C05467=1049.152,167.646,409.024,171.137,36.035,156.777
C05468=1049.158,167.895,409.001,171.139,36.037,156.778
C05469=1049.163,168.144,408.978,171.141,36.039,156.778
C05470=1049.169,168.392,408.955,171.143,36.041,156.778
C05471=1049.176,168.641,408.932,171.145,36.043,156.779
C05472=1049.181,168.890,408.909,171.148,36.046,156.779
C05473=1049.187,169.139,408.886,171.150,36.047,156.780
C05474=1049.194,169.388,408.862,171.152,36.050,156.780
C05475=1049.199,169.637,408.839,171.154,36.052,156.780
C05476=1049.205,169.886,408.817,171.157,36.054,156.781
C05477=1049.212,170.134,408.794,171.159,36.056,156.781
C05478=1049.217,170.383,408.771,171.161,36.058,156.782
C05479=1049.223,170.632,408.748,171.163,36.060,156.782
C05480=1049.229,170.881,408.725,171.165,36.062,156.783
C05481=1049.235,171.131,408.702,171.168,36.065,156.783
C05482=1049.241,171.379,408.678,171.170,36.067,156.783
C05483=1049.248,171.627,408.656,171.172,36.069,156.784
C05484=1049.253,171.876,408.633,171.174,36.071,156.784
C05485=1049.259,172.125,408.610,171.176,36.073,156.785
C05486=1049.265,172.374,408.587,171.179,36.075,156.785
C05487=1049.271,172.624,408.564,171.181,36.077,156.785
C05488=1049.277,172.872,408.540,171.183,36.080,156.786
C05489=1049.283,173.121,408.517,171.185,36.081,156.786
C05490=1049.289,173.369,408.495,171.188,36.084,156.787
C05491=1049.296,173.654,408.468,171.190,36.086,156.787
C05492=1049.303,173.939,408.442,171.193,36.089,156.788
C05493=1049.310,174.224,408.415,171.195,36.091,156.788
C05494=1049.317,174.508,408.388,171.198,36.094,156.789
C05495=1049.324,174.758,408.366,171.200,36.096,156.789
C05496=1049.329,175.007,408.343,171.202,36.097,156.789
C05497=1049.335,175.255,408.319,171.204,36.100,156.790
C05498=1049.341,175.504,408.296,171.206,36.102,156.790
C05499=1049.347,175.753,408.273,171.209,36.104,156.791
C05500=1049.353,176.002,408.249,171.211,36.106,156.791
C05501=1049.359,176.250,408.226,171.213,36.108,156.791
C05502=1049.365,176.499,408.203,171.216,36.110,156.792
C05503=1049.372,176.748,408.180,171.219,36.113,156.792
C05504=1049.378,176.997,408.157,171.221,36.115,156.793
C05505=1049.384,177.246,408.134,171.223,36.117,156.793
C05506=1049.390,177.495,408.110,171.225,36.119,156.794
C05507=1049.396,177.744,408.087,171.227,36.121,156.794
C05508=1049.402,177.992,408.063,171.230,36.123,156.794
C05509=1049.408,178.242,408.040,171.232,36.125,156.795
C05510=1049.414,178.490,408.017,171.234,36.128,156.795
C05511=1049.420,178.739,407.993,171.236,36.129,156.796
C05512=1049.427,178.988,407.970,171.239,36.132,156.796
C05513=1049.433,179.237,407.946,171.241,36.134,156.796
C05514=1049.439,179.485,407.924,171.243,36.136,156.797
C05515=1049.446,179.734,407.900,171.245,36.138,156.797
C05516=1049.451,179.983,407.877,171.247,36.140,156.798
C05517=1049.457,180.231,407.853,171.251,36.142,156.798
C05518=1049.464,180.481,407.830,171.253,36.145,156.799
C05519=1049.470,180.729,407.806,171.255,36.147,156.799
C05520=1049.476,180.979,407.783,171.257,36.149,156.799
C05521=1049.482,181.227,407.759,171.260,36.151,156.800
C05522=1049.488,181.476,407.736,171.262,36.153,156.800
C05523=1049.495,181.725,407.712,171.264,36.155,156.801
C05524=1049.501,181.973,407.689,171.266,36.158,156.801
C05525=1049.507,182.223,407.665,171.268,36.159,156.801
C05526=1049.513,182.471,407.642,171.272,36.162,156.802
C05527=1049.519,182.721,407.618,171.274,36.164,156.802
C05528=1049.526,182.969,407.595,171.276,36.166,156.803
C05529=1049.532,183.217,407.572,171.278,36.168,156.803
C05530=1049.538,183.467,407.548,171.281,36.170,156.804
C05531=1049.545,183.715,407.525,171.283,36.172,156.804
C05532=1049.551,183.964,407.501,171.285,36.175,156.804
C05533=1049.556,184.213,407.477,171.287,36.177,156.805
C05534=1049.563,184.462,407.453,171.290,36.179,156.805
C05535=1049.568,184.711,407.429,171.293,36.181,156.806
C05536=1049.574,184.959,407.405,171.295,36.184,156.806
C05537=1049.580,185.209,407.381,171.297,36.186,156.807
C05538=1049.586,185.457,407.358,171.300,36.188,156.807
C05539=1049.592,185.705,407.334,171.302,36.191,156.808
C05540=1049.598,185.955,407.309,171.304,36.193,156.808
C05541=1049.604,186.203,407.286,171.306,36.196,156.809
C05542=1049.609,186.451,407.261,171.309,36.197,156.809
C05543=1049.615,186.701,407.238,171.311,36.200,156.809
C05544=1049.621,186.950,407.214,171.313,36.202,156.810
C05545=1049.627,187.199,407.190,171.315,36.205,156.810
C05546=1049.633,187.447,407.166,171.319,36.207,156.811
C05547=1049.639,187.696,407.142,171.321,36.209,156.811
C05548=1049.645,187.945,407.117,171.323,36.211,156.812
C05549=1049.651,188.193,407.094,171.325,36.214,156.812
C05550=1049.656,188.442,407.069,171.328,36.216,156.813
C05551=1049.663,188.691,407.045,171.330,36.219,156.813
C05552=1049.668,188.940,407.021,171.332,36.221,156.814
C05553=1049.674,189.188,406.997,171.334,36.223,156.814
C05554=1049.680,189.438,406.972,171.338,36.226,156.815
C05555=1049.687,189.722,406.945,171.340,36.229,156.815
C05556=1049.694,190.006,406.918,171.342,36.231,156.816
C05557=1049.701,190.290,406.890,171.345,36.233,156.816
C05558=1049.708,190.575,406.863,171.348,36.236,156.817
C05559=1049.713,190.823,406.839,171.351,36.239,156.817
C05560=1049.720,191.072,406.815,171.353,36.241,156.818
C05561=1049.725,191.321,406.790,171.356,36.243,156.818
C05562=1049.732,191.570,406.766,171.358,36.246,156.819
C05563=1049.737,191.818,406.741,171.360,36.248,156.819
C05564=1049.744,192.067,406.717,171.362,36.251,156.820
C05565=1049.749,192.316,406.693,171.366,36.253,156.820
C05566=1049.756,192.564,406.669,171.368,36.255,156.820
C05567=1049.762,192.814,406.645,171.370,36.257,156.821
C05568=1049.768,193.062,406.621,171.372,36.260,156.821
C05569=1049.774,193.311,406.596,171.375,36.262,156.822
C05570=1049.779,193.560,406.572,171.377,36.265,156.822
C05571=1049.786,193.808,406.547,171.380,36.267,156.823
C05572=1049.791,194.057,406.523,171.382,36.269,156.823
C05573=1049.798,194.306,406.499,171.385,36.272,156.824
C05574=1049.804,194.555,406.474,171.387,36.274,156.824
C05575=1049.810,194.803,406.451,171.389,36.276,156.825
C05576=1049.816,195.052,406.425,171.392,36.279,156.825
C05577=1049.822,195.300,406.402,171.395,36.281,156.826
C05578=1049.828,195.550,406.377,171.397,36.283,156.826
C05579=1049.834,195.799,406.353,171.399,36.286,156.827
C05580=1049.840,196.047,406.328,171.402,36.288,156.827
C05581=1049.846,196.296,406.303,171.405,36.291,156.828
C05582=1049.853,196.545,406.279,171.407,36.293,156.828
C05583=1049.858,196.793,406.255,171.409,36.296,156.829
C05584=1049.865,197.042,406.230,171.412,36.297,156.829
C05585=1049.870,197.290,406.206,171.415,36.300,156.829
C05586=1049.877,197.539,406.182,171.417,36.302,156.830
C05587=1049.883,197.788,406.157,171.419,36.305,156.830
C05588=1049.889,198.037,406.132,171.422,36.307,156.831
C05589=1049.895,198.286,406.109,171.424,36.310,156.831
C05590=1049.901,198.534,406.083,171.427,36.312,156.832
C05591=1049.908,198.783,406.059,171.430,36.314,156.832
C05592=1049.913,199.031,406.034,171.432,36.317,156.833
C05593=1049.920,199.280,406.010,171.434,36.319,156.833
C05594=1049.926,199.530,405.986,171.437,36.322,156.834
C05595=1049.932,199.777,405.961,171.440,36.324,156.834
C05596=1049.938,200.026,405.937,171.442,36.327,156.835
C05597=1049.944,200.275,405.911,171.445,36.329,156.835
C05598=1049.951,200.524,405.887,171.447,36.331,156.836
C05599=1049.957,200.772,405.862,171.450,36.333,156.836
C05600=1049.962,201.021,405.838,171.452,36.336,156.837
C05601=1049.969,201.270,405.813,171.455,36.338,156.837
C05602=1049.975,201.519,405.788,171.458,36.341,156.838
C05603=1049.982,201.768,405.763,171.460,36.343,156.838
C05604=1049.987,202.016,405.739,171.462,36.346,156.839
C05605=1049.993,202.265,405.713,171.465,36.348,156.839
C05606=1050.000,202.514,405.689,171.468,36.351,156.840
C05607=1050.005,202.762,405.664,171.470,36.353,156.840
C05608=1050.011,203.011,405.639,171.472,36.356,156.841
C05609=1050.017,203.260,405.614,171.476,36.358,156.841
C05610=1050.024,203.509,405.589,171.478,36.361,156.842
C05611=1050.029,203.757,405.565,171.480,36.364,156.842
C05612=1050.035,204.006,405.539,171.483,36.366,156.843
C05613=1050.041,204.254,405.514,171.486,36.368,156.843
C05614=1050.048,204.503,405.489,171.488,36.371,156.844
C05615=1050.053,204.752,405.464,171.490,36.373,156.844
C05616=1050.059,205.000,405.439,171.494,36.376,156.845
C05617=1050.065,205.249,405.414,171.496,36.379,156.845
C05618=1050.072,205.498,405.390,171.498,36.381,156.846
C05619=1050.097,206.550,405.283,171.730,36.477,156.865
C05620=1050.104,206.804,405.256,171.731,36.481,156.866
C05621=1050.111,207.059,405.230,171.733,36.485,156.867
C05622=1050.118,207.314,405.204,171.736,36.488,156.867
C05623=1050.124,207.567,405.177,171.737,36.491,156.868
C05624=1050.131,207.816,405.150,171.740,36.495,156.869
C05625=1050.137,208.065,405.125,171.742,36.498,156.870
C05626=1050.143,208.313,405.098,171.744,36.501,156.870
C05627=1050.150,208.562,405.072,171.746,36.504,156.871
C05628=1050.156,208.811,405.046,171.747,36.508,156.872
C05629=1050.162,209.060,405.019,171.750,36.511,156.872
C05630=1050.169,209.308,404.993,171.751,36.515,156.873
C05631=1050.175,209.556,404.967,171.754,36.518,156.874
C05632=1050.182,209.805,404.940,171.756,36.521,156.874
C05633=1050.188,210.053,404.915,171.757,36.525,156.875
C05634=1050.194,210.301,404.889,171.760,36.528,156.876
C05635=1050.201,210.551,404.862,171.762,36.531,156.876
C05636=1050.207,210.799,404.836,171.764,36.534,156.877
C05637=1050.214,211.047,404.809,171.766,36.538,156.878
C05638=1050.220,211.296,404.783,171.767,36.541,156.878
C05639=1050.226,211.544,404.757,171.770,36.545,156.879
C05640=1050.233,211.793,404.730,171.772,36.548,156.880
C05641=1050.239,212.041,404.704,171.774,36.551,156.881
C05642=1050.246,212.290,404.678,171.776,36.554,156.881
C05643=1050.252,212.539,404.651,171.778,36.558,156.882
C05644=1050.258,212.787,404.625,171.780,36.561,156.883
C05645=1050.265,213.036,404.598,171.782,36.564,156.883
C05646=1050.271,213.284,404.571,171.784,36.568,156.884
C05647=1050.278,213.533,404.545,171.786,36.571,156.885
C05648=1050.284,213.781,404.518,171.789,36.575,156.885
C05649=1050.290,214.029,404.492,171.790,36.577,156.886
C05650=1050.297,214.278,404.465,171.792,36.581,156.887
C05651=1050.303,214.526,404.439,171.795,36.584,156.887
C05652=1050.310,214.775,404.412,171.796,36.588,156.888
C05653=1050.316,215.023,404.386,171.799,36.591,156.889
C05654=1050.322,215.272,404.359,171.801,36.594,156.890
C05655=1050.328,215.521,404.333,171.803,36.598,156.890
C05656=1050.335,215.770,404.306,171.805,36.601,156.891
C05657=1050.341,216.018,404.279,171.807,36.604,156.892
C05658=1050.348,216.266,404.253,171.809,36.607,156.892
C05659=1050.354,216.515,404.226,171.811,36.611,156.893
C05660=1050.360,216.763,404.200,171.814,36.614,156.894
C05661=1050.367,217.012,404.173,171.815,36.618,156.894
C05662=1050.373,217.260,404.146,171.817,36.621,156.895
C05663=1050.380,217.509,404.120,171.820,36.624,156.896
C05664=1050.386,217.757,404.093,171.821,36.627,156.896
C05665=1050.393,218.006,404.067,171.824,36.630,156.897
C05666=1050.399,218.255,404.039,171.826,36.634,156.898
C05667=1050.406,218.502,404.013,171.828,36.637,156.898
C05668=1050.413,218.751,403.986,171.830,36.640,156.899
C05669=1050.418,219.000,403.959,171.832,36.643,156.900
C05670=1050.425,219.248,403.933,171.835,36.647,156.901
C05671=1050.431,219.497,403.906,171.836,36.650,156.901
C05672=1050.439,219.745,403.879,171.839,36.653,156.902
C05673=1050.444,219.993,403.852,171.841,36.656,156.903
C05674=1050.451,220.242,403.825,171.842,36.659,156.903
C05675=1050.458,220.491,403.799,171.845,36.663,156.904
C05676=1050.464,220.751,403.771,171.847,36.667,156.905
C05677=1050.471,221.011,403.743,171.850,36.670,156.905
C05678=1050.478,221.271,403.714,171.852,36.673,156.906
C05679=1050.484,221.530,403.686,171.854,36.677,156.907
C05680=1050.491,221.779,403.659,171.856,36.680,156.907
C05681=1050.496,222.028,403.632,171.859,36.683,156.908
C05682=1050.503,222.276,403.604,171.861,36.686,156.909
C05683=1050.510,222.524,403.578,171.862,36.690,156.910
C05684=1050.516,222.773,403.550,171.865,36.693,156.910
C05685=1050.522,223.021,403.524,171.867,36.696,156.911
C05686=1050.528,223.270,403.497,171.869,36.699,156.912
C05687=1050.535,223.519,403.469,171.871,36.703,156.912
C05688=1050.541,223.767,403.442,171.874,36.706,156.913
C05689=1050.548,224.015,403.415,171.876,36.709,156.914
C05690=1050.554,224.263,403.389,171.877,36.712,156.914
C05691=1050.561,224.512,403.361,171.880,36.716,156.915
C05692=1050.567,224.761,403.334,171.882,36.719,156.916
C05693=1050.573,225.009,403.306,171.885,36.723,156.916
C05694=1050.580,225.258,403.279,171.887,36.726,156.917
C05695=1050.586,225.506,403.252,171.889,36.729,156.918
C05696=1050.592,225.755,403.225,171.891,36.732,156.918
C05697=1050.599,226.003,403.197,171.893,36.736,156.919
C05698=1050.606,226.252,403.171,171.896,36.739,156.920
C05699=1050.612,226.499,403.144,171.897,36.742,156.920
C05700=1050.618,226.749,403.117,171.900,36.745,156.921
C05701=1050.625,226.997,403.089,171.902,36.748,156.922
C05702=1050.631,227.245,403.061,171.905,36.752,156.923
C05703=1050.637,227.494,403.034,171.907,36.755,156.923
C05704=1050.644,227.742,403.007,171.908,36.758,156.924
C05705=1050.650,227.991,402.980,171.911,36.761,156.925
C05706=1050.657,228.239,402.952,171.913,36.764,156.925
C05707=1050.664,228.487,402.925,171.916,36.768,156.926
C05708=1050.670,228.736,402.898,171.918,36.771,156.927
C05709=1050.676,228.984,402.871,171.921,36.774,156.927
C05710=1050.683,229.232,402.843,171.922,36.777,156.928
C05711=1050.689,229.481,402.816,171.924,36.780,156.929
C05712=1050.695,229.729,402.788,171.927,36.784,156.929
C05713=1050.701,229.978,402.760,171.929,36.787,156.930
C05714=1050.708,230.226,402.733,171.932,36.790,156.931
C05715=1050.715,230.475,402.705,171.933,36.793,156.931
C05716=1050.721,230.723,402.678,171.936,36.797,156.932
C05717=1050.727,230.972,402.651,171.938,36.800,156.933
C05718=1050.734,231.220,402.623,171.941,36.804,156.934
C05719=1050.740,231.468,402.595,171.943,36.806,156.934
C05720=1050.747,231.716,402.568,171.945,36.809,156.935
C05721=1050.752,231.966,402.540,171.947,36.813,156.936
C05722=1050.759,232.214,402.512,171.949,36.816,156.936
C05723=1050.766,232.462,402.485,171.952,36.820,156.937
C05724=1050.772,232.710,402.457,171.954,36.823,156.938
C05725=1050.779,232.959,402.430,171.957,36.826,156.938
C05726=1050.785,233.207,402.402,171.959,36.829,156.939
C05727=1050.791,233.456,402.373,171.962,36.833,156.940
C05728=1050.797,233.704,402.346,171.963,36.836,156.940
C05729=1050.804,233.952,402.318,171.965,36.839,156.941
C05730=1050.811,234.200,402.291,171.968,36.842,156.942
C05731=1050.817,234.449,402.262,171.970,36.846,156.943
C05732=1050.823,234.702,402.235,171.973,36.849,156.943
C05733=1050.829,234.954,402.207,171.975,36.852,156.944
C05734=1050.836,235.206,402.178,171.978,36.855,156.945
C05735=1050.842,235.459,402.150,171.980,36.859,156.945
C05736=1050.849,235.707,402.122,171.982,36.862,156.946
C05737=1050.855,235.956,402.094,171.984,36.865,156.947
C05738=1050.862,236.204,402.066,171.986,36.868,156.947
C05739=1050.868,236.453,402.038,171.989,36.871,156.948
C05740=1050.874,236.701,402.011,171.991,36.875,156.949
C05741=1050.881,236.949,401.983,171.994,36.878,156.949
C05742=1050.887,237.198,401.955,171.996,36.881,156.950
C05743=1050.893,237.446,401.927,171.999,36.884,156.951
C05744=1050.900,237.695,401.899,172.001,36.888,156.951
C05745=1050.907,237.942,401.871,172.004,36.891,156.952
C05746=1050.913,238.191,401.842,172.006,36.894,156.953
C05747=1050.920,238.440,401.815,172.007,36.897,156.954
C05748=1050.926,238.687,401.787,172.010,36.900,156.954
C05749=1050.932,238.936,401.759,172.012,36.904,156.955
C05750=1050.938,239.185,401.731,172.015,36.907,156.956
C05751=1050.945,239.432,401.703,172.017,36.910,156.956
C05752=1050.951,239.681,401.675,172.020,36.913,156.957
C05753=1050.958,239.930,401.647,172.022,36.916,156.958
C05754=1050.965,240.178,401.619,172.025,36.920,156.958
C05755=1050.971,240.427,401.591,172.027,36.923,156.959
C05756=1050.977,240.675,401.562,172.029,36.926,156.960
C05757=1050.983,240.923,401.534,172.032,36.929,156.960
C05758=1050.990,241.172,401.506,172.034,36.932,156.961
C05759=1050.997,241.420,401.478,172.037,36.936,156.962
C05760=1051.003,241.668,401.450,172.039,36.939,156.962
C05761=1051.009,241.916,401.422,172.042,36.942,156.963
C05762=1051.015,242.164,401.393,172.044,36.945,156.964
C05763=1051.022,242.413,401.365,172.047,36.948,156.964
C05764=1051.028,242.661,401.337,172.049,36.952,156.965
C05765=1051.034,242.910,401.308,172.051,36.955,156.966
C05766=1051.041,243.158,401.280,172.053,36.958,156.967
C05767=1051.047,243.406,401.251,172.056,36.961,156.967
C05768=1051.054,243.655,401.224,172.058,36.965,156.968
C05769=1051.060,243.903,401.195,172.060,36.968,156.969
C05770=1051.066,244.151,401.166,172.063,36.971,156.969
C05771=1051.073,244.400,401.138,172.065,36.974,156.970
C05772=1051.079,244.648,401.109,172.068,36.978,156.971
C05773=1051.086,244.896,401.082,172.070,36.981,156.971
C05774=1051.092,245.145,401.053,172.073,36.984,156.972
C05775=1051.098,245.393,401.024,172.075,36.987,156.973
C05776=1051.105,245.641,400.996,172.078,36.990,156.973
C05777=1051.111,245.890,400.968,172.080,36.994,156.974
C05778=1051.117,246.138,400.938,172.083,36.996,156.975
C05779=1051.123,246.386,400.909,172.085,37.000,156.976
C05780=1051.130,246.635,400.882,172.088,37.004,156.976
C05781=1051.136,246.883,400.853,172.090,37.006,156.977
C05782=1051.142,247.131,400.824,172.093,37.010,156.978
C05783=1051.148,247.380,400.795,172.095,37.013,156.978
C05784=1051.155,247.628,400.766,172.097,37.017,156.979
C05785=1051.161,247.876,400.737,172.100,37.019,156.980
C05786=1051.168,248.124,400.709,172.102,37.023,156.981
C05787=1051.174,248.372,400.680,172.105,37.026,156.981
C05788=1051.179,248.620,400.652,172.107,37.029,156.982
C05789=1051.186,248.867,400.624,172.110,37.032,156.983
C05790=1051.192,249.114,400.594,172.112,37.036,156.983
C05791=1051.198,249.362,400.565,172.115,37.039,156.984
C05792=1051.204,249.609,400.537,172.117,37.042,156.985
C05793=1051.211,249.857,400.508,172.120,37.045,156.985
C05794=1051.217,250.104,400.480,172.122,37.049,156.986
C05795=1051.224,250.352,400.450,172.125,37.052,156.987
C05796=1051.230,250.600,400.421,172.127,37.055,156.988
C05797=1051.236,250.849,400.393,172.131,37.058,156.988
C05798=1051.243,251.096,400.364,172.133,37.062,156.989
C05799=1051.249,251.345,400.335,172.136,37.065,156.990
C05800=1051.255,251.593,400.306,172.138,37.068,156.990
C05801=1051.262,251.841,400.277,172.140,37.071,156.991
C05802=1051.268,252.089,400.248,172.143,37.075,156.992
C05803=1051.274,252.337,400.219,172.145,37.078,156.993
C05804=1051.281,252.587,400.191,172.148,37.081,156.993
C05805=1051.287,252.835,400.162,172.150,37.084,156.994
C05806=1051.293,253.083,400.133,172.153,37.088,156.995
C05807=1051.300,253.331,400.104,172.155,37.091,156.995
C05808=1051.306,253.579,400.075,172.158,37.094,156.996
C05809=1051.313,253.827,400.046,172.160,37.097,156.997
C05810=1051.319,254.075,400.017,172.164,37.101,156.998
C05811=1051.326,254.324,399.988,172.166,37.104,156.998
C05812=1051.332,254.572,399.959,172.169,37.107,156.999
C05813=1051.338,254.820,399.929,172.171,37.110,157.000
C05814=1051.344,255.068,399.900,172.174,37.114,157.000
C05815=1051.351,255.316,399.871,172.176,37.116,157.001
C05816=1051.358,255.565,399.842,172.179,37.119,157.002
C05817=1051.364,255.813,399.813,172.181,37.123,157.002
C05818=1051.370,256.061,399.784,172.184,37.126,157.003
C05819=1051.377,256.309,399.755,172.187,37.129,157.004
C05820=1051.384,256.558,399.725,172.190,37.132,157.004
C05821=1051.390,256.806,399.696,172.192,37.136,157.005
C05822=1051.397,257.054,399.667,172.195,37.139,157.006
C05823=1051.403,257.302,399.638,172.197,37.142,157.007
C05824=1051.410,257.551,399.609,172.200,37.145,157.007
C05825=1051.416,257.799,399.580,172.202,37.148,157.008
C05826=1051.422,258.047,399.551,172.205,37.152,157.009
C05827=1051.429,258.295,399.521,172.208,37.155,157.009
C05828=1051.436,258.543,399.492,172.210,37.158,157.010
C05829=1051.442,258.791,399.463,172.213,37.161,157.011
C05830=1051.448,259.040,399.433,172.215,37.165,157.012
C05831=1051.455,259.288,399.404,172.218,37.167,157.012
C05832=1051.462,259.536,399.374,172.221,37.171,157.013
C05833=1051.468,259.784,399.345,172.224,37.174,157.014
C05834=1051.475,260.033,399.316,172.226,37.177,157.014
C05835=1051.481,260.281,399.287,172.229,37.180,157.015
C05836=1051.488,260.529,399.257,172.231,37.183,157.016
C05837=1051.494,260.777,399.228,172.235,37.187,157.016
C05838=1051.501,261.026,399.199,172.237,37.190,157.017
C05839=1051.507,261.273,399.169,172.240,37.193,157.018
C05840=1051.514,261.522,399.139,172.242,37.196,157.019
C05841=1051.520,261.770,399.110,172.245,37.199,157.019
C05842=1051.527,262.018,399.080,172.248,37.203,157.020
C05843=1051.534,262.266,399.051,172.251,37.205,157.021
C05844=1051.540,262.513,399.022,172.253,37.208,157.021
C05845=1051.547,262.759,398.993,172.256,37.212,157.022
C05846=1051.553,263.005,398.964,172.259,37.215,157.023
C05847=1051.559,263.252,398.934,172.262,37.218,157.023
C05848=1051.566,263.498,398.905,172.264,37.221,157.024
C05849=1051.573,263.746,398.875,172.267,37.225,157.025
C05850=1051.579,263.992,398.846,172.269,37.228,157.026
C05851=1051.585,264.239,398.815,172.273,37.231,157.026
C05852=1051.591,264.487,398.786,172.275,37.235,157.027
C05853=1051.598,264.734,398.757,172.278,37.238,157.028
C05854=1051.604,264.983,398.726,172.280,37.241,157.028
C05855=1051.611,265.231,398.697,172.283,37.244,157.029
C05856=1051.618,265.479,398.667,172.286,37.247,157.030
C05857=1051.623,265.728,398.637,172.289,37.250,157.031
C05858=1051.630,265.975,398.607,172.291,37.254,157.031
C05859=1051.637,266.223,398.577,172.294,37.257,157.032
C05860=1051.642,266.472,398.548,172.297,37.260,157.033
C05861=1051.650,266.720,398.517,172.300,37.264,157.034
C05862=1051.656,266.967,398.488,172.302,37.267,157.034
C05863=1051.662,267.217,398.458,172.305,37.270,157.035
C05864=1051.669,267.464,398.428,172.308,37.273,157.036
C05865=1051.675,267.712,398.398,172.311,37.277,157.036
C05866=1051.682,267.960,398.367,172.313,37.280,157.037
C05867=1051.688,268.208,398.338,172.316,37.283,157.038
C05868=1051.694,268.457,398.308,172.319,37.286,157.039
C05869=1051.701,268.704,398.278,172.322,37.289,157.039
C05870=1051.707,268.953,398.247,172.324,37.293,157.040
C05871=1051.714,269.200,398.217,172.328,37.296,157.041
C05872=1051.720,269.449,398.187,172.330,37.299,157.041
C05873=1051.727,269.697,398.158,172.333,37.303,157.042
C05874=1051.733,269.945,398.127,172.335,37.306,157.043
C05875=1051.740,270.193,398.097,172.339,37.309,157.044
C05876=1051.746,270.442,398.067,172.341,37.313,157.044
C05877=1051.753,270.689,398.037,172.344,37.316,157.045
C05878=1051.759,270.938,398.006,172.347,37.319,157.046
C05879=1051.766,271.185,397.976,172.350,37.322,157.047
C05880=1051.772,271.434,397.946,172.353,37.325,157.047
C05881=1051.779,271.681,397.916,172.356,37.329,157.048
C05882=1051.785,271.930,397.885,172.359,37.332,157.049
C05883=1051.792,272.177,397.855,172.361,37.335,157.049
C05884=1051.798,272.426,397.825,172.365,37.339,157.050
C05885=1051.804,272.673,397.794,172.367,37.342,157.051
C05886=1051.811,272.922,397.764,172.370,37.345,157.052
C05887=1051.817,273.169,397.734,172.373,37.349,157.052
C05888=1051.823,273.418,397.703,172.376,37.352,157.053
C05889=1051.830,273.666,397.673,172.378,37.355,157.054
C05890=1051.836,273.914,397.643,172.382,37.359,157.055
C05891=1051.843,274.163,397.612,172.384,37.361,157.055
C05892=1051.849,274.410,397.582,172.387,37.365,157.056
C05893=1051.856,274.659,397.551,172.390,37.368,157.057
C05894=1051.861,274.906,397.521,172.393,37.371,157.058
C05895=1051.869,275.154,397.490,172.395,37.375,157.058
C05896=1051.875,275.403,397.460,172.399,37.378,157.059
C05897=1051.881,275.650,397.429,172.401,37.381,157.060
C05898=1051.887,275.899,397.398,172.404,37.385,157.061
C05899=1051.894,276.146,397.368,172.408,37.388,157.061
C05900=1051.900,276.396,397.337,172.410,37.392,157.062
C05901=1051.907,276.644,397.306,172.414,37.394,157.063
C05902=1051.914,276.894,397.275,172.416,37.398,157.064
C05903=1051.920,277.143,397.245,172.419,37.401,157.064
C05904=1051.927,277.391,397.214,172.422,37.404,157.065
C05905=1051.933,277.639,397.183,172.425,37.408,157.066
C05906=1051.940,277.887,397.153,172.427,37.411,157.067
C05907=1051.946,278.135,397.123,172.431,37.415,157.067
C05908=1051.953,278.383,397.091,172.433,37.418,157.068
C05909=1051.959,278.631,397.061,172.437,37.421,157.069
C05910=1051.965,278.879,397.029,172.440,37.425,157.070
C05911=1051.972,279.127,396.999,172.442,37.427,157.070
C05912=1051.978,279.375,396.969,172.446,37.431,157.071
C05913=1051.985,279.623,396.938,172.448,37.434,157.072
C05914=1051.991,279.871,396.907,172.452,37.438,157.073
C05915=1051.997,280.119,396.876,172.454,37.441,157.073
C05916=1052.004,280.367,396.845,172.458,37.444,157.074
C05917=1052.011,280.615,396.814,172.460,37.448,157.075
C05918=1052.017,280.864,396.783,172.463,37.451,157.076
C05919=1052.023,281.111,396.752,172.467,37.455,157.076
C05920=1052.030,281.359,396.721,172.469,37.458,157.077
C05921=1052.036,281.607,396.690,172.473,37.461,157.078
C05922=1052.042,281.854,396.659,172.475,37.464,157.079
C05923=1052.049,282.103,396.628,172.479,37.468,157.079
C05924=1052.056,282.351,396.596,172.481,37.471,157.080
C05925=1052.062,282.599,396.566,172.484,37.475,157.081
C05926=1052.068,282.847,396.535,172.487,37.478,157.082
C05927=1052.075,283.094,396.503,172.490,37.481,157.082
C05928=1052.081,283.343,396.472,172.493,37.485,157.083
C05929=1052.088,283.591,396.441,172.496,37.488,157.084
C05930=1052.094,283.838,396.410,172.500,37.492,157.085
C05931=1052.101,284.086,396.379,172.502,37.495,157.086
C05932=1052.107,284.335,396.348,172.506,37.498,157.086
C05933=1052.114,284.582,396.316,172.508,37.501,157.087
C05934=1052.121,284.830,396.285,172.512,37.505,157.088
C05935=1052.127,285.078,396.254,172.514,37.508,157.089
C05936=1052.133,285.326,396.223,172.518,37.512,157.089
C05937=1052.139,285.574,396.191,172.521,37.515,157.090
C05938=1052.146,285.822,396.160,172.524,37.519,157.091
C05939=1052.153,286.070,396.128,172.527,37.522,157.092
C05940=1052.159,286.318,396.097,172.530,37.525,157.092
C05941=1052.165,286.566,396.067,172.533,37.528,157.093
C05942=1052.172,286.814,396.035,172.536,37.532,157.094
C05943=1052.179,287.062,396.004,172.539,37.535,157.095
C05944=1052.185,287.310,395.972,172.543,37.539,157.096
C05945=1052.192,287.557,395.941,172.545,37.542,157.096
C05946=1052.199,287.805,395.909,172.549,37.545,157.097
C05947=1052.206,288.053,395.878,172.551,37.549,157.098
C05948=1052.212,288.301,395.846,172.555,37.552,157.099
C05949=1052.218,288.549,395.814,172.557,37.555,157.099
C05950=1052.224,288.797,395.783,172.561,37.559,157.100
C05951=1052.231,289.044,395.752,172.564,37.562,157.101
C05952=1052.237,289.293,395.720,172.567,37.566,157.102
C05953=1052.244,289.541,395.689,172.570,37.569,157.103
C05954=1052.251,289.788,395.657,172.573,37.573,157.103
C05955=1052.257,290.036,395.626,172.577,37.576,157.104
C05956=1052.267,290.423,395.576,172.582,37.581,157.105
C05957=1052.277,290.809,395.527,172.587,37.587,157.107
C05958=1052.287,291.195,395.477,172.592,37.592,157.108
C05959=1052.297,291.581,395.427,172.597,37.597,157.109
C05960=1052.308,291.951,395.380,172.601,37.603,157.110
C05961=1052.317,292.321,395.333,172.605,37.608,157.111
C05962=1052.327,292.691,395.285,172.610,37.613,157.113
C05963=1052.337,293.061,395.238,172.615,37.618,157.114
C05964=1052.343,293.309,395.206,172.619,37.621,157.115
C05965=1052.350,293.557,395.174,172.621,37.625,157.115
C05966=1052.357,293.805,395.142,172.625,37.628,157.116
C05967=1052.363,294.053,395.110,172.628,37.632,157.117
C05968=1052.369,294.301,395.079,172.631,37.635,157.118
C05969=1052.376,294.548,395.046,172.635,37.639,157.119
C05970=1052.382,294.796,395.014,172.637,37.642,157.119
C05971=1052.389,295.044,394.982,172.641,37.646,157.120
C05972=1052.395,295.292,394.950,172.644,37.649,157.121
C05973=1052.402,295.540,394.919,172.647,37.653,157.122
C05974=1052.408,295.787,394.886,172.651,37.656,157.123
C05975=1052.415,296.035,394.855,172.654,37.660,157.124
C05976=1052.422,296.283,394.822,172.657,37.663,157.124
C05977=1052.427,296.531,394.790,172.661,37.667,157.125
C05978=1052.435,296.778,394.758,172.663,37.670,157.126
C05979=1052.441,297.026,394.725,172.667,37.674,157.127
C05980=1052.447,297.274,394.693,172.670,37.678,157.128
C05981=1052.453,297.522,394.660,172.673,37.681,157.128
C05982=1052.460,297.770,394.629,172.677,37.685,157.129
C05983=1052.466,298.017,394.596,172.680,37.688,157.130
C05984=1052.472,298.265,394.563,172.683,37.692,157.131
C05985=1052.478,298.513,394.531,172.687,37.695,157.132
C05986=1052.485,298.761,394.498,172.689,37.699,157.133
C05987=1052.492,299.009,394.466,172.693,37.703,157.134
C05988=1052.499,299.256,394.433,172.697,37.706,157.134
C05989=1052.505,299.504,394.401,172.699,37.709,157.135
C05990=1052.511,299.752,394.368,172.703,37.713,157.136
C05991=1052.517,300.000,394.336,172.707,37.717,157.137
C05992=1052.524,300.247,394.304,172.709,37.720,157.138
C05993=1052.530,300.495,394.272,172.713,37.724,157.139
C05994=1052.536,300.743,394.239,172.717,37.728,157.139
C05995=1052.543,300.990,394.206,172.719,37.731,157.140
C05996=1052.550,301.239,394.173,172.723,37.735,157.141
C05997=1052.557,301.486,394.141,172.727,37.739,157.142
C05998=1052.563,301.733,394.108,172.729,37.742,157.143
C05999=1052.569,301.981,394.075,172.733,37.746,157.144
C06000=1052.575,302.229,394.043,172.736,37.749,157.144
C06001=1052.582,302.477,394.010,172.740,37.753,157.145
C06002=1052.588,302.725,393.977,172.743,37.757,157.146
C06003=1052.596,302.972,393.945,172.746,37.760,157.147
C06004=1052.602,303.220,393.913,172.750,37.764,157.148
C06005=1052.608,303.468,393.880,172.753,37.768,157.149
C06006=1052.615,303.716,393.847,172.756,37.771,157.150
C06007=1052.621,303.963,393.814,172.760,37.774,157.150
C06008=1052.629,304.239,393.778,172.764,37.778,157.151
C06009=1052.636,304.516,393.741,172.767,37.782,157.152
C06010=1052.643,304.793,393.704,172.771,37.787,157.153
C06011=1052.651,305.069,393.668,172.775,37.791,157.154
C06012=1052.657,305.316,393.635,172.779,37.794,157.155
C06013=1052.664,305.565,393.602,172.782,37.798,157.156
C06014=1052.670,305.812,393.569,172.786,37.802,157.157
C06015=1052.677,306.059,393.536,172.789,37.805,157.158
C06016=1052.684,306.308,393.503,172.792,37.809,157.159
C06017=1052.690,306.555,393.470,172.796,37.812,157.159
C06018=1052.697,306.802,393.438,172.800,37.816,157.160
C06019=1052.704,307.051,393.405,172.803,37.820,157.161
C06020=1052.711,307.298,393.371,172.806,37.823,157.162
C06021=1052.717,307.545,393.339,172.810,37.827,157.163
C06022=1052.724,307.794,393.305,172.813,37.831,157.164
C06023=1052.730,308.041,393.273,172.817,37.834,157.164
C06024=1052.737,308.289,393.239,172.821,37.838,157.165
C06025=1052.744,308.536,393.206,172.823,37.841,157.166
C06026=1052.750,308.784,393.173,172.827,37.845,157.167
C06027=1052.758,309.032,393.141,172.831,37.849,157.168
C06028=1052.764,309.279,393.107,172.834,37.853,157.169
C06029=1052.771,309.527,393.074,172.838,37.856,157.170
C06030=1052.778,309.774,393.041,172.842,37.860,157.171
C06031=1052.785,310.023,393.008,172.844,37.863,157.171
C06032=1052.791,310.270,392.975,172.848,37.867,157.172
C06033=1052.798,310.518,392.941,172.852,37.871,157.173
C06034=1052.804,310.765,392.908,172.855,37.874,157.174
C06035=1052.812,311.013,392.875,172.859,37.878,157.175
C06036=1052.818,311.261,392.842,172.863,37.882,157.176
C06037=1052.825,311.508,392.808,172.866,37.885,157.177
C06038=1052.831,311.756,392.775,172.870,37.889,157.178
C06039=1052.839,312.004,392.741,172.873,37.893,157.178
C06040=1052.845,312.251,392.709,172.876,37.896,157.179
C06041=1052.852,312.499,392.675,172.880,37.900,157.180
C06042=1052.859,312.747,392.642,172.884,37.904,157.181
C06043=1052.866,312.994,392.609,172.888,37.908,157.182
C06044=1052.872,313.242,392.575,172.891,37.911,157.183
C06045=1052.879,313.489,392.542,172.895,37.915,157.184
C06046=1052.886,313.737,392.508,172.899,37.919,157.185
C06047=1052.892,313.985,392.475,172.901,37.923,157.186
C06048=1052.899,314.233,392.441,172.905,37.927,157.187
C06049=1052.905,314.480,392.407,172.909,37.931,157.187
C06050=1052.912,314.728,392.373,172.913,37.934,157.188
C06051=1052.918,314.975,392.339,172.916,37.938,157.189
C06052=1052.925,315.223,392.306,172.920,37.942,157.190
C06053=1052.931,315.470,392.272,172.924,37.946,157.191
C06054=1052.938,315.718,392.238,172.928,37.950,157.192
C06055=1052.944,315.965,392.204,172.930,37.954,157.193
C06056=1052.951,316.213,392.170,172.934,37.957,157.194
C06057=1052.957,316.460,392.136,172.938,37.961,157.195
C06058=1052.964,316.708,392.102,172.941,37.965,157.196
C06059=1052.970,316.956,392.068,172.945,37.969,157.197
C06060=1052.977,317.203,392.034,172.949,37.973,157.198
C06061=1052.983,317.452,392.001,172.953,37.977,157.199
C06062=1052.990,317.699,391.967,172.957,37.981,157.200
C06063=1052.996,317.947,391.933,172.960,37.985,157.200
C06064=1053.004,318.228,391.894,172.964,37.989,157.201
C06065=1053.011,318.508,391.855,172.968,37.993,157.203
C06066=1053.019,318.788,391.817,172.973,37.998,157.204
C06067=1053.027,319.069,391.778,172.977,38.002,157.205
C06068=1053.033,319.317,391.743,172.980,38.006,157.206
C06069=1053.040,319.564,391.710,172.984,38.010,157.207
C06070=1053.046,319.812,391.675,172.988,38.014,157.208
C06071=1053.053,320.060,391.642,172.992,38.018,157.208
C06072=1053.060,320.308,391.607,172.995,38.022,157.209
C06073=1053.067,320.555,391.574,172.999,38.026,157.210
C06074=1053.073,320.803,391.539,173.003,38.030,157.211
C06075=1053.080,321.050,391.504,173.007,38.034,157.212
C06076=1053.087,321.298,391.470,173.010,38.038,157.213
C06077=1053.093,321.545,391.436,173.014,38.042,157.214
C06078=1053.100,321.793,391.402,173.018,38.046,157.215
C06079=1053.107,322.040,391.367,173.022,38.049,157.216
C06080=1053.114,322.288,391.333,173.026,38.053,157.217
C06081=1053.120,322.536,391.299,173.029,38.057,157.218
C06082=1053.126,322.783,391.265,173.033,38.061,157.219
C06083=1053.134,323.030,391.230,173.037,38.065,157.220
C06084=1053.140,323.278,391.196,173.041,38.069,157.221
C06085=1053.148,323.525,391.161,173.044,38.073,157.222
C06086=1053.154,323.773,391.127,173.048,38.077,157.223
C06087=1053.161,324.021,391.093,173.052,38.081,157.224
C06088=1053.168,324.268,391.058,173.056,38.085,157.225
C06089=1053.174,324.515,391.024,173.059,38.089,157.226
C06090=1053.182,324.762,390.989,173.063,38.093,157.227
C06091=1053.188,325.010,390.955,173.067,38.097,157.228
C06092=1053.195,325.258,390.921,173.072,38.101,157.229
C06093=1053.202,325.505,390.886,173.076,38.105,157.230
C06094=1053.209,325.753,390.852,173.079,38.109,157.231
C06095=1053.216,326.000,390.817,173.083,38.113,157.232
C06096=1053.223,326.248,390.782,173.087,38.117,157.232
C06097=1053.229,326.496,390.748,173.091,38.121,157.233
C06098=1053.237,326.743,390.713,173.095,38.125,157.234
C06099=1053.243,326.991,390.679,173.098,38.129,157.235
C06100=1053.250,327.238,390.644,173.102,38.133,157.236
C06101=1053.257,327.485,390.609,173.106,38.137,157.237
C06102=1053.264,327.733,390.575,173.111,38.141,157.238
C06103=1053.271,327.980,390.539,173.115,38.145,157.239
C06104=1053.278,328.228,390.506,173.118,38.149,157.240
C06105=1053.285,328.476,390.470,173.122,38.153,157.241
C06106=1053.291,328.723,390.435,173.126,38.157,157.242
C06107=1053.299,328.970,390.401,173.130,38.161,157.243
C06108=1053.305,329.218,390.366,173.134,38.165,157.244
C06109=1053.313,329.466,390.331,173.139,38.169,157.245
C06110=1053.320,329.713,390.296,173.142,38.173,157.246
C06111=1053.327,329.960,390.261,173.146,38.177,157.247
C06112=1053.334,330.208,390.226,173.150,38.181,157.248
C06113=1053.341,330.455,390.191,173.154,38.185,157.249
C06114=1053.347,330.703,390.156,173.158,38.190,157.250
C06115=1053.354,330.950,390.121,173.161,38.194,157.251
C06116=1053.361,331.198,390.086,173.166,38.198,157.252
C06117=1053.367,331.445,390.051,173.170,38.202,157.253
C06118=1053.374,331.693,390.016,173.174,38.207,157.255
C06119=1053.381,331.940,389.981,173.178,38.210,157.255
C06120=1053.388,332.215,389.941,173.183,38.215,157.257
C06121=1053.396,332.491,389.902,173.187,38.220,157.258
C06122=1053.404,332.766,389.863,173.192,38.225,157.259
C06123=1053.411,333.041,389.823,173.196,38.229,157.260
C06124=1053.419,333.289,389.788,173.200,38.234,157.261
C06125=1053.426,333.537,389.753,173.204,38.238,157.262
C06126=1053.432,333.784,389.717,173.208,38.242,157.263
C06127=1053.439,334.032,389.682,173.212,38.246,157.264
C06128=1053.446,334.279,389.647,173.216,38.251,157.265
C06129=1053.452,334.526,389.611,173.220,38.255,157.266
C06130=1053.460,334.774,389.575,173.225,38.259,157.267
C06131=1053.466,335.021,389.540,173.229,38.263,157.269
C06132=1053.473,335.269,389.505,173.233,38.268,157.270
C06133=1053.480,335.516,389.469,173.236,38.272,157.271
C06134=1053.488,335.764,389.434,173.241,38.276,157.272
C06135=1053.494,336.011,389.398,173.245,38.280,157.273
C06136=1053.501,336.258,389.363,173.249,38.284,157.274
C06137=1053.508,336.505,389.327,173.253,38.289,157.275
C06138=1053.515,336.753,389.291,173.258,38.293,157.276
C06139=1053.522,337.000,389.256,173.262,38.298,157.277
C06140=1053.529,337.248,389.220,173.266,38.302,157.278
C06141=1053.535,337.495,389.184,173.270,38.306,157.279
C06142=1053.542,337.743,389.148,173.274,38.310,157.280
C06143=1053.549,337.989,389.113,173.278,38.315,157.281
C06144=1053.555,338.237,389.077,173.282,38.319,157.282
C06145=1053.563,338.485,389.041,173.287,38.324,157.284
C06146=1053.570,338.732,389.006,173.291,38.328,157.285
C06147=1053.576,338.979,388.969,173.295,38.333,157.286
C06148=1053.584,339.226,388.933,173.299,38.337,157.287
C06149=1053.591,339.474,388.898,173.304,38.341,157.288
C06150=1053.597,339.721,388.861,173.308,38.346,157.289
C06151=1053.605,339.968,388.825,173.312,38.350,157.290
C06152=1053.611,340.216,388.790,173.317,38.355,157.291
C06153=1053.618,340.463,388.753,173.321,38.359,157.292
C06154=1053.625,340.710,388.717,173.325,38.364,157.294
C06155=1053.632,340.957,388.682,173.330,38.368,157.295
C06156=1053.639,341.205,388.645,173.334,38.372,157.296
C06157=1053.646,341.452,388.609,173.337,38.377,157.297
C06158=1053.653,341.700,388.573,173.342,38.381,157.298
C06159=1053.660,341.946,388.537,173.346,38.386,157.299
C06160=1053.668,342.195,388.501,173.350,38.390,157.300
C06161=1053.674,342.442,388.465,173.355,38.395,157.301
C06162=1053.682,342.689,388.429,173.359,38.399,157.302
C06163=1053.688,342.936,388.392,173.364,38.403,157.304
C06164=1053.696,343.184,388.356,173.368,38.408,157.305
C06165=1053.702,343.431,388.320,173.372,38.413,157.306
C06166=1053.709,343.677,388.284,173.377,38.417,157.307
C06167=1053.716,343.925,388.247,173.381,38.422,157.308
C06168=1053.723,344.172,388.211,173.385,38.426,157.309
C06169=1053.730,344.420,388.174,173.390,38.431,157.310
C06170=1053.737,344.667,388.137,173.394,38.435,157.312
C06171=1053.744,344.914,388.102,173.399,38.440,157.313
C06172=1053.751,345.162,388.065,173.403,38.445,157.314
C06173=1053.758,345.409,388.029,173.407,38.449,157.315
C06174=1053.765,345.656,387.991,173.412,38.454,157.316
C06175=1053.772,345.903,387.955,173.416,38.459,157.317
C06176=1053.780,346.174,387.914,173.421,38.464,157.319
C06177=1053.787,346.446,387.875,173.426,38.468,157.320
C06178=1053.795,346.717,387.835,173.431,38.473,157.321
C06179=1053.803,346.988,387.795,173.435,38.479,157.323
C06180=1053.810,347.236,387.758,173.440,38.483,157.324
C06181=1053.816,347.482,387.721,173.444,38.488,157.325
C06182=1053.824,347.730,387.685,173.449,38.493,157.326
C06183=1053.831,347.978,387.648,173.453,38.498,157.327
C06184=1053.838,348.224,387.611,173.458,38.502,157.328
C06185=1053.844,348.472,387.574,173.462,38.507,157.330
C06186=1053.852,348.719,387.537,173.467,38.511,157.331
C06187=1053.859,348.966,387.500,173.471,38.516,157.332
C06188=1053.866,349.214,387.464,173.476,38.521,157.333
C06189=1053.873,349.461,387.426,173.481,38.526,157.334
C06190=1053.881,349.708,387.390,173.486,38.531,157.336
C06191=1053.887,349.955,387.353,173.490,38.535,157.337
C06192=1053.894,350.202,387.316,173.495,38.540,157.338
C06193=1053.901,350.449,387.278,173.499,38.545,157.339
C06194=1053.909,350.696,387.241,173.504,38.549,157.340
C06195=1053.916,350.943,387.205,173.508,38.554,157.342
C06196=1053.923,351.190,387.167,173.513,38.559,157.343
C06197=1053.930,351.438,387.131,173.517,38.564,157.344
C06198=1053.937,351.685,387.093,173.522,38.568,157.345
C06199=1053.944,351.932,387.056,173.526,38.573,157.347
C06200=1053.951,352.179,387.018,173.531,38.578,157.348
C06201=1053.958,352.427,386.982,173.535,38.583,157.349
C06202=1053.965,352.674,386.944,173.540,38.588,157.350
C06203=1053.973,352.921,386.907,173.544,38.593,157.352
C06204=1053.979,353.167,386.869,173.549,38.598,157.353
C06205=1053.986,353.415,386.832,173.555,38.602,157.354
C06206=1053.994,353.662,386.794,173.559,38.607,157.355
C06207=1054.001,353.909,386.758,173.564,38.612,157.357
C06208=1054.008,354.157,386.720,173.568,38.617,157.358
C06209=1054.015,354.404,386.682,173.573,38.622,157.359
C06210=1054.022,354.650,386.645,173.578,38.627,157.360
C06211=1054.029,354.897,386.608,173.582,38.632,157.362
C06212=1054.036,355.144,386.570,173.587,38.637,157.363
C06213=1054.043,355.392,386.533,173.591,38.642,157.364
C06214=1054.051,355.639,386.495,173.596,38.647,157.365
C06215=1054.058,355.886,386.458,173.602,38.652,157.367
C06216=1054.065,356.133,386.420,173.606,38.657,157.368
C06217=1054.073,356.379,386.382,173.611,38.662,157.369
C06218=1054.080,356.627,386.344,173.616,38.667,157.371
C06219=1054.087,356.874,386.307,173.620,38.672,157.372
C06220=1054.094,357.121,386.269,173.625,38.677,157.373
C06221=1054.102,357.368,386.232,173.630,38.682,157.374
C06222=1054.109,357.615,386.194,173.635,38.687,157.376
C06223=1054.117,357.862,386.156,173.640,38.692,157.377
C06224=1054.124,358.109,386.119,173.645,38.697,157.378
C06225=1054.131,358.356,386.081,173.649,38.702,157.380
C06226=1054.138,358.603,386.043,173.654,38.707,157.381
C06227=1054.145,358.850,386.005,173.659,38.712,157.382
C06228=1054.152,359.097,385.967,173.664,38.718,157.384
C06229=1054.160,359.343,385.929,173.669,38.723,157.385
C06230=1054.166,359.591,385.891,173.674,38.727,157.386
C06231=1054.174,359.838,385.853,173.678,38.733,157.388
C06232=1054.182,360.114,385.811,173.684,38.738,157.389
C06233=1054.191,360.391,385.767,173.690,38.744,157.391
C06234=1054.198,360.667,385.725,173.695,38.750,157.392
C06235=1054.207,360.943,385.682,173.700,38.756,157.394
C06236=1054.214,361.190,385.645,173.706,38.761,157.395
C06237=1054.221,361.438,385.606,173.711,38.766,157.396
C06238=1054.229,361.685,385.568,173.715,38.772,157.398
C06239=1054.236,361.931,385.530,173.720,38.777,157.399
C06240=1054.243,362.178,385.491,173.725,38.782,157.400
C06241=1054.250,362.425,385.454,173.731,38.787,157.402
C06242=1054.258,362.672,385.415,173.735,38.792,157.403
C06243=1054.265,362.919,385.376,173.740,38.798,157.405
C06244=1054.273,363.166,385.338,173.745,38.803,157.406
C06245=1054.280,363.413,385.300,173.751,38.809,157.407
C06246=1054.287,363.660,385.261,173.755,38.813,157.409
C06247=1054.294,363.906,385.223,173.760,38.819,157.410
C06248=1054.302,364.154,385.184,173.765,38.824,157.412
C06249=1054.309,364.400,385.146,173.771,38.830,157.413
C06250=1054.316,364.647,385.107,173.776,38.835,157.414
C06251=1054.323,364.894,385.068,173.780,38.841,157.416
C06252=1054.331,365.141,385.029,173.785,38.846,157.417
C06253=1054.338,365.388,384.991,173.791,38.851,157.419
C06254=1054.345,365.635,384.952,173.796,38.857,157.420
C06255=1054.352,365.881,384.914,173.801,38.862,157.421
C06256=1054.360,366.129,384.875,173.807,38.868,157.423
C06257=1054.367,366.376,384.836,173.811,38.873,157.424
C06258=1054.375,366.622,384.798,173.816,38.878,157.426
C06259=1054.382,366.870,384.759,173.821,38.884,157.427
C06260=1054.389,367.116,384.720,173.827,38.889,157.429
C06261=1054.397,367.362,384.681,173.832,38.895,157.430
C06262=1054.404,367.610,384.642,173.837,38.901,157.432
C06263=1054.412,367.856,384.603,173.843,38.906,157.433
C06264=1054.419,368.104,384.564,173.848,38.911,157.434
C06265=1054.426,368.350,384.525,173.853,38.917,157.436
C06266=1054.434,368.597,384.486,173.858,38.922,157.437
C06267=1054.441,368.844,384.447,173.863,38.928,157.439
C06268=1054.449,369.090,384.408,173.868,38.934,157.440
C06269=1054.457,369.338,384.369,173.874,38.939,157.442
C06270=1054.463,369.584,384.330,173.879,38.944,157.443
C06271=1054.472,369.831,384.291,173.884,38.950,157.445
C06272=1054.479,370.078,384.252,173.890,38.956,157.446
C06273=1054.486,370.325,384.212,173.895,38.962,157.448
C06274=1054.494,370.571,384.174,173.900,38.967,157.449
C06275=1054.502,370.818,384.134,173.906,38.972,157.451
C06276=1054.509,371.065,384.096,173.911,38.978,157.452
C06277=1054.517,371.311,384.056,173.917,38.984,157.454
C06278=1054.524,371.558,384.016,173.922,38.990,157.455
C06279=1054.532,371.805,383.978,173.927,38.995,157.457
C06280=1054.540,372.052,383.938,173.933,39.001,157.458
C06281=1054.547,372.298,383.898,173.938,39.007,157.460
C06282=1054.554,372.546,383.859,173.943,39.012,157.461
C06283=1054.562,372.792,383.819,173.949,39.018,157.463
C06284=1054.569,373.039,383.780,173.954,39.024,157.464
C06285=1054.576,373.285,383.740,173.960,39.030,157.466
C06286=1054.584,373.532,383.700,173.965,39.035,157.467
C06287=1054.592,373.779,383.661,173.971,39.041,157.469
C06288=1054.600,374.074,383.613,173.977,39.048,157.471
C06289=1054.610,374.368,383.566,173.984,39.055,157.473
C06290=1054.619,374.664,383.519,173.990,39.062,157.475
C06291=1054.628,374.959,383.471,173.997,39.069,157.476
C06292=1054.635,375.206,383.431,174.002,39.075,157.478
C06293=1054.642,375.452,383.391,174.007,39.081,157.480
C06294=1054.650,375.699,383.351,174.013,39.087,157.481
C06295=1054.658,375.946,383.311,174.019,39.093,157.483
C06296=1054.666,376.193,383.271,174.025,39.099,157.484
C06297=1054.673,376.439,383.232,174.030,39.105,157.486
C06298=1054.680,376.686,383.192,174.036,39.111,157.488
C06299=1054.688,376.932,383.151,174.041,39.117,157.489
C06300=1054.696,377.179,383.111,174.047,39.123,157.491
C06301=1054.703,377.425,383.072,174.052,39.129,157.492
C06302=1054.711,377.672,383.032,174.058,39.135,157.494
C06303=1054.719,377.918,382.991,174.064,39.141,157.496
C06304=1054.727,378.165,382.951,174.070,39.147,157.497
C06305=1054.735,378.412,382.911,174.075,39.153,157.499
C06306=1054.743,378.659,382.871,174.081,39.159,157.500
C06307=1054.750,378.905,382.831,174.087,39.165,157.502
C06308=1054.758,379.151,382.791,174.092,39.171,157.504
C06309=1054.765,379.398,382.751,174.099,39.178,157.506
C06310=1054.773,379.644,382.710,174.104,39.184,157.507
C06311=1054.781,379.891,382.670,174.110,39.189,157.509
C06312=1054.789,380.137,382.629,174.115,39.196,157.510
C06313=1054.797,380.384,382.590,174.121,39.202,157.512
C06314=1054.804,380.631,382.548,174.127,39.208,157.514
C06315=1054.812,380.878,382.508,174.133,39.215,157.516
C06316=1054.820,381.124,382.468,174.139,39.220,157.517
C06317=1054.827,381.371,382.427,174.144,39.227,157.519
C06318=1054.835,381.617,382.386,174.151,39.233,157.521
C06319=1054.843,381.864,382.346,174.156,39.240,157.522
C06320=1054.850,382.111,382.305,174.162,39.246,157.524
C06321=1054.858,382.357,382.264,174.168,39.252,157.526
C06322=1054.866,382.603,382.223,174.174,39.258,157.527
C06323=1054.874,382.850,382.182,174.180,39.265,157.529
C06324=1054.882,383.096,382.142,174.186,39.271,157.531
C06325=1054.889,383.343,382.100,174.191,39.278,157.533
C06326=1054.897,383.589,382.060,174.198,39.284,157.534
C06327=1054.905,383.835,382.019,174.204,39.290,157.536
C06328=1054.912,384.082,381.978,174.209,39.297,157.538
C06329=1054.920,384.328,381.937,174.216,39.303,157.540
C06330=1054.928,384.574,381.897,174.221,39.309,157.541
C06331=1054.936,384.821,381.855,174.227,39.316,157.543
C06332=1054.944,385.067,381.815,174.234,39.322,157.545
C06333=1054.951,385.314,381.773,174.240,39.329,157.547
C06334=1054.960,385.561,381.733,174.245,39.336,157.548
C06335=1054.968,385.806,381.691,174.252,39.342,157.550
C06336=1054.975,386.053,381.650,174.258,39.348,157.552
C06337=1054.983,386.299,381.609,174.263,39.355,157.554
C06338=1054.991,386.547,381.568,174.270,39.362,157.556
C06339=1054.999,386.792,381.526,174.276,39.368,157.557
C06340=1055.007,387.039,381.486,174.283,39.375,157.559
C06341=1055.015,387.285,381.444,174.288,39.381,157.561
C06342=1055.024,387.531,381.403,174.295,39.388,157.563
C06343=1055.031,387.778,381.362,174.301,39.394,157.565
C06344=1055.042,388.104,381.306,174.309,39.403,157.567
C06345=1055.052,388.432,381.252,174.317,39.412,157.570
C06346=1055.063,388.759,381.197,174.326,39.421,157.572
C06347=1055.074,389.086,381.142,174.334,39.430,157.575
C06348=1055.082,389.333,381.101,174.340,39.436,157.576
C06349=1055.090,389.579,381.059,174.347,39.443,157.578
C06350=1055.098,389.824,381.017,174.353,39.450,157.580
C06351=1055.106,390.072,380.976,174.359,39.457,157.582
C06352=1055.114,390.318,380.934,174.365,39.464,157.584
C06353=1055.123,390.564,380.892,174.372,39.470,157.586
C06354=1055.130,390.810,380.850,174.378,39.477,157.588
C06355=1055.138,391.056,380.808,174.385,39.484,157.589
C06356=1055.147,391.302,380.766,174.391,39.491,157.591
C06357=1055.154,391.549,380.725,174.397,39.498,157.593
C06358=1055.162,391.796,380.683,174.403,39.505,157.595
C06359=1055.170,392.041,380.641,174.410,39.512,157.597
C06360=1055.179,392.288,380.599,174.417,39.519,157.599
C06361=1055.186,392.534,380.557,174.423,39.526,157.601
C06362=1055.195,392.780,380.515,174.430,39.532,157.603
C06363=1055.202,393.026,380.473,174.436,39.540,157.605
C06364=1055.212,393.272,380.431,174.443,39.547,157.607
C06365=1055.219,393.518,380.389,174.450,39.554,157.609
C06366=1055.227,393.765,380.346,174.456,39.561,157.611
C06367=1055.235,394.012,380.304,174.463,39.568,157.613
C06368=1055.243,394.257,380.261,174.469,39.575,157.615
C06369=1055.252,394.504,380.219,174.475,39.582,157.617
C06370=1055.259,394.750,380.177,174.482,39.589,157.619
C06371=1055.267,394.996,380.135,174.488,39.596,157.621
C06372=1055.277,395.242,380.092,174.495,39.604,157.623
C06373=1055.284,395.488,380.050,174.502,39.610,157.625
C06374=1055.293,395.734,380.007,174.508,39.618,157.627
C06375=1055.301,395.981,379.965,174.515,39.625,157.629
C06376=1055.309,396.227,379.922,174.522,39.633,157.631
C06377=1055.317,396.473,379.880,174.529,39.639,157.633
C06378=1055.326,396.719,379.837,174.535,39.647,157.635
C06379=1055.334,396.965,379.795,174.542,39.654,157.637
C06380=1055.342,397.211,379.752,174.549,39.661,157.639
C06381=1055.351,397.458,379.709,174.556,39.669,157.641
C06382=1055.358,397.703,379.667,174.563,39.676,157.643
C06383=1055.367,397.950,379.624,174.570,39.684,157.645
C06384=1055.375,398.196,379.581,174.577,39.691,157.647
C06385=1055.384,398.442,379.538,174.584,39.698,157.650
C06386=1055.392,398.688,379.495,174.590,39.706,157.652
C06387=1055.400,398.935,379.452,174.597,39.713,157.654
C06388=1055.408,399.181,379.409,174.604,39.721,157.656
C06389=1055.416,399.426,379.366,174.611,39.728,157.658
C06390=1055.425,399.672,379.323,174.618,39.736,157.660
C06391=1055.433,399.918,379.280,174.624,39.743,157.662
C06392=1055.442,400.164,379.237,174.632,39.751,157.665
C06393=1055.450,400.410,379.194,174.639,39.758,157.667
C06394=1055.458,400.657,379.150,174.646,39.766,157.669
C06395=1055.466,400.903,379.107,174.653,39.774,157.671
C06396=1055.475,401.149,379.064,174.660,39.781,157.673
C06397=1055.484,401.396,379.021,174.667,39.789,157.675
C06398=1055.493,401.642,378.978,174.675,39.797,157.678
C06399=1055.501,401.887,378.934,174.681,39.804,157.680
C06400=1055.513,402.233,378.873,174.691,39.815,157.683
C06401=1055.524,402.577,378.813,174.701,39.826,157.686
C06402=1055.536,402.922,378.751,174.711,39.837,157.689
C06403=1055.548,403.266,378.691,174.721,39.848,157.692
C06404=1055.557,403.513,378.647,174.729,39.856,157.694
C06405=1055.565,403.759,378.603,174.736,39.863,157.697
C06406=1055.574,404.004,378.559,174.743,39.871,157.699
C06407=1055.582,404.251,378.516,174.751,39.879,157.701
C06408=1055.590,404.496,378.472,174.758,39.887,157.704
C06409=1055.600,404.743,378.428,174.765,39.895,157.706
C06410=1055.608,404.989,378.384,174.773,39.903,157.708
C06411=1055.616,405.234,378.340,174.780,39.911,157.710
C06412=1055.625,405.481,378.296,174.787,39.919,157.713
C06413=1055.634,405.727,378.253,174.795,39.927,157.715
C06414=1055.642,405.972,378.208,174.802,39.935,157.717
C06415=1055.650,406.219,378.164,174.809,39.944,157.720
C06416=1055.659,406.464,378.120,174.818,39.951,157.722
C06417=1055.667,406.710,378.075,174.825,39.960,157.724
C06418=1055.677,406.956,378.031,174.833,39.968,157.727
C06419=1055.685,407.202,377.987,174.840,39.976,157.729
C06420=1055.693,407.448,377.943,174.847,39.984,157.731
C06421=1055.702,407.694,377.899,174.855,39.992,157.734
C06422=1055.710,407.939,377.854,174.862,40.001,157.736
C06423=1055.719,408.186,377.810,174.870,40.009,157.739
C06424=1055.728,408.431,377.766,174.878,40.017,157.741
C06425=1055.736,408.678,377.721,174.886,40.025,157.744
C06426=1055.746,408.923,377.677,174.893,40.034,157.746
C06427=1055.754,409.169,377.632,174.901,40.042,157.748
C06428=1055.762,409.415,377.588,174.909,40.050,157.751
C06429=1055.772,409.661,377.543,174.917,40.059,157.753
C06430=1055.781,409.907,377.498,174.924,40.067,157.756
C06431=1055.789,410.153,377.454,174.932,40.076,157.758
C06432=1055.798,410.398,377.409,174.940,40.084,157.761
C06433=1055.807,410.644,377.364,174.948,40.093,157.763
C06434=1055.815,410.890,377.320,174.956,40.101,157.766
C06435=1055.825,411.136,377.275,174.964,40.110,157.768
C06436=1055.834,411.382,377.230,174.972,40.118,157.771
C06437=1055.843,411.628,377.185,174.979,40.127,157.773
C06438=1055.852,411.873,377.140,174.988,40.135,157.776
C06439=1055.860,412.119,377.096,174.996,40.144,157.778
C06440=1055.869,412.365,377.050,175.003,40.153,157.781
C06441=1055.878,412.611,377.005,175.012,40.161,157.783
C06442=1055.888,412.856,376.960,175.019,40.169,157.786
C06443=1055.896,413.102,376.916,175.028,40.178,157.788
C06444=1055.905,413.348,376.870,175.036,40.187,157.791
C06445=1055.914,413.594,376.825,175.045,40.196,157.794
C06446=1055.924,413.839,376.780,175.052,40.204,157.796
C06447=1055.933,414.085,376.735,175.061,40.213,157.799
C06448=1055.942,414.331,376.689,175.069,40.222,157.801
C06449=1055.950,414.577,376.643,175.078,40.231,157.804
C06450=1055.959,414.823,376.598,175.085,40.240,157.807
C06451=1055.968,415.068,376.552,175.094,40.249,157.809
C06452=1055.977,415.314,376.506,175.102,40.258,157.812
C06453=1055.986,415.560,376.461,175.111,40.267,157.815
C06454=1055.995,415.806,376.415,175.119,40.276,157.817
C06455=1056.004,416.051,376.369,175.127,40.285,157.820
C06456=1056.017,416.402,376.305,175.139,40.298,157.824
C06457=1056.030,416.752,376.239,175.152,40.311,157.828
C06458=1056.043,417.102,376.174,175.164,40.324,157.832
C06459=1056.057,417.453,376.108,175.176,40.337,157.836
C06460=1056.065,417.699,376.062,175.185,40.346,157.838
C06461=1056.074,417.944,376.016,175.193,40.355,157.841
C06462=1056.083,418.190,375.971,175.202,40.364,157.844
C06463=1056.093,418.436,375.924,175.211,40.374,157.847
C06464=1056.103,418.681,375.878,175.220,40.383,157.849
C06465=1056.112,418.927,375.833,175.228,40.392,157.852
C06466=1056.121,419.172,375.787,175.236,40.401,157.855
C06467=1056.131,419.418,375.740,175.246,40.411,157.858
C06468=1056.140,419.663,375.694,175.255,40.420,157.861
C06469=1056.149,419.908,375.648,175.263,40.430,157.864
C06470=1056.158,420.155,375.601,175.272,40.439,157.866
C06471=1056.168,420.400,375.555,175.281,40.449,157.869
C06472=1056.177,420.645,375.509,175.290,40.458,157.872
C06473=1056.186,420.891,375.461,175.299,40.468,157.875
C06474=1056.195,421.136,375.415,175.308,40.477,157.878
C06475=1056.205,421.382,375.369,175.317,40.487,157.881
C06476=1056.214,421.627,375.321,175.326,40.497,157.884
C06477=1056.223,421.872,375.275,175.334,40.506,157.887
C06478=1056.233,422.119,375.228,175.344,40.516,157.890
C06479=1056.242,422.363,375.181,175.353,40.526,157.893
C06480=1056.252,422.609,375.135,175.362,40.536,157.896
C06481=1056.261,422.854,375.087,175.371,40.545,157.899
C06482=1056.271,423.100,375.041,175.380,40.555,157.902
C06483=1056.280,423.345,374.994,175.390,40.565,157.905
C06484=1056.290,423.591,374.947,175.399,40.575,157.908
C06485=1056.299,423.835,374.900,175.408,40.585,157.911
C06486=1056.308,424.082,374.853,175.418,40.594,157.914
C06487=1056.318,424.327,374.806,175.428,40.604,157.917
C06488=1056.328,424.571,374.759,175.437,40.615,157.920
C06489=1056.338,424.817,374.711,175.446,40.624,157.923
C06490=1056.347,425.063,374.665,175.456,40.634,157.926
C06491=1056.356,425.308,374.617,175.465,40.644,157.929
C06492=1056.366,425.553,374.570,175.475,40.655,157.932
C06493=1056.376,425.799,374.522,175.485,40.664,157.935
C06494=1056.386,426.044,374.475,175.494,40.675,157.938
C06495=1056.396,426.290,374.427,175.504,40.685,157.942
C06496=1056.405,426.534,374.380,175.513,40.695,157.945
C06497=1056.415,426.780,374.332,175.523,40.705,157.948
C06498=1056.424,427.025,374.285,175.533,40.715,157.951
C06499=1056.435,427.270,374.237,175.543,40.726,157.954
C06500=1056.444,427.516,374.189,175.552,40.736,157.957
C06501=1056.453,427.761,374.141,175.563,40.747,157.961
C06502=1056.464,428.006,374.093,175.572,40.757,157.964
C06503=1056.473,428.251,374.046,175.582,40.768,157.967
C06504=1056.483,428.495,373.998,175.593,40.778,157.970
C06505=1056.493,428.741,373.950,175.602,40.788,157.974
C06506=1056.503,428.986,373.901,175.612,40.799,157.977
C06507=1056.512,429.232,373.854,175.622,40.809,157.980
C06508=1056.523,429.477,373.805,175.632,40.820,157.984
C06509=1056.533,429.722,373.757,175.643,40.831,157.987
C06510=1056.542,429.968,373.709,175.653,40.841,157.990
C06511=1056.553,430.212,373.661,175.663,40.852,157.994
C06512=1056.563,430.470,373.610,175.674,40.863,157.997
C06513=1056.573,430.728,373.558,175.684,40.874,158.001
C06514=1056.583,430.986,373.507,175.695,40.886,158.004
C06515=1056.593,431.243,373.457,175.706,40.897,158.008
C06516=1056.604,431.489,373.408,175.717,40.908,158.011
C06517=1056.614,431.733,373.360,175.727,40.919,158.015
C06518=1056.624,431.978,373.311,175.738,40.930,158.018
C06519=1056.634,432.223,373.263,175.748,40.941,158.022
C06520=1056.645,432.468,373.213,175.758,40.952,158.025
C06521=1056.654,432.713,373.165,175.769,40.963,158.029
C06522=1056.664,432.958,373.116,175.780,40.974,158.032
C06523=1056.674,433.203,373.067,175.791,40.985,158.036
C06524=1056.690,433.563,372.995,175.806,41.001,158.041
C06525=1056.704,433.923,372.923,175.822,41.018,158.046
C06526=1056.719,434.282,372.851,175.838,41.034,158.051
C06527=1056.735,434.641,372.779,175.854,41.051,158.057
C06528=1056.744,434.886,372.730,175.865,41.062,158.060
C06529=1056.755,435.131,372.680,175.876,41.073,158.064
C06530=1056.765,435.376,372.631,175.887,41.085,158.068
C06531=1056.776,435.621,372.582,175.898,41.096,158.071
C06532=1056.786,435.865,372.532,175.909,41.107,158.075
C06533=1056.797,436.110,372.483,175.921,41.119,158.079
C06534=1056.807,436.355,372.433,175.932,41.131,158.082
C06535=1056.817,436.600,372.384,175.943,41.142,158.086
C06536=1056.828,436.845,372.334,175.954,41.154,158.090
C06537=1056.839,437.090,372.285,175.965,41.165,158.094
C06538=1056.849,437.335,372.235,175.977,41.177,158.097
C06539=1056.859,437.579,372.185,175.988,41.189,158.101
C06540=1056.870,437.824,372.135,175.999,41.200,158.105
C06541=1056.880,438.069,372.085,176.012,41.212,158.109
C06542=1056.891,438.314,372.036,176.023,41.224,158.113
C06543=1056.901,438.558,371.985,176.034,41.236,158.117
C06544=1056.912,438.802,371.935,176.046,41.248,158.121
C06545=1056.922,439.047,371.885,176.057,41.260,158.124
C06546=1056.933,439.292,371.835,176.070,41.271,158.128
C06547=1056.943,439.537,371.785,176.081,41.284,158.132
C06548=1056.954,439.782,371.734,176.093,41.296,158.136
C06549=1056.965,440.026,371.684,176.105,41.308,158.140
C06550=1056.975,440.271,371.633,176.117,41.320,158.144
C06551=1056.986,440.515,371.583,176.129,41.332,158.148
C06552=1056.997,440.760,371.532,176.141,41.344,158.152
C06553=1057.007,441.004,371.482,176.153,41.356,158.156
C06554=1057.018,441.249,371.431,176.165,41.369,158.160
C06555=1057.029,441.494,371.380,176.177,41.381,158.164
C06556=1057.040,441.738,371.330,176.189,41.393,158.168
C06557=1057.051,441.983,371.279,176.202,41.406,158.172
C06558=1057.062,442.227,371.228,176.214,41.418,158.177
C06559=1057.073,442.472,371.177,176.226,41.430,158.181
C06560=1057.083,442.716,371.126,176.238,41.443,158.185
C06561=1057.094,442.960,371.075,176.251,41.456,158.189
C06562=1057.105,443.205,371.023,176.264,41.468,158.193
C06563=1057.116,443.450,370.973,176.276,41.481,158.197
C06564=1057.127,443.694,370.921,176.289,41.494,158.202
C06565=1057.139,443.938,370.870,176.302,41.506,158.206
C06566=1057.149,444.183,370.819,176.314,41.519,158.210
C06567=1057.161,444.427,370.768,176.327,41.532,158.214
C06568=1057.170,444.645,370.722,176.338,41.543,158.218
C06569=1057.180,444.863,370.676,176.350,41.555,158.222
C06570=1057.190,445.081,370.629,176.361,41.566,158.226
C06571=1057.200,445.298,370.584,176.373,41.578,158.230
C06572=1057.210,445.517,370.538,176.384,41.589,158.234
C06573=1057.220,445.734,370.491,176.396,41.601,158.238
C06574=1057.230,445.952,370.445,176.407,41.612,158.242
C06575=1057.241,446.170,370.400,176.419,41.624,158.245
C06576=1057.252,446.414,370.348,176.432,41.637,158.250
C06577=1057.263,446.657,370.296,176.445,41.650,158.254
C06578=1057.274,446.901,370.245,176.459,41.664,158.259
C06579=1057.287,447.144,370.193,176.472,41.677,158.263
C06580=1057.299,447.388,370.143,176.486,41.689,158.268
C06581=1057.313,447.631,370.093,176.499,41.701,158.272
C06582=1057.328,447.876,370.043,176.513,41.714,158.276
C06583=1057.343,448.120,369.995,176.526,41.726,158.280
C06584=1057.360,448.364,369.947,176.540,41.738,158.285
C06585=1057.377,448.609,369.899,176.554,41.749,158.289
C06586=1057.395,448.853,369.852,176.568,41.761,158.293
C06587=1057.414,449.098,369.806,176.581,41.772,158.297
C06588=1057.433,449.344,369.759,176.596,41.783,158.301
C06589=1057.453,449.589,369.714,176.610,41.794,158.305
C06590=1057.475,449.834,369.669,176.624,41.805,158.309
C06591=1057.497,450.079,369.626,176.639,41.815,158.312
C06592=1057.171,450.095,369.340,176.635,41.922,158.342
C06593=1057.148,449.850,369.385,176.621,41.912,158.339
C06594=1057.128,449.604,369.429,176.607,41.901,158.335
C06595=1057.107,449.359,369.475,176.592,41.890,158.331
C06596=1057.087,449.114,369.520,176.578,41.879,158.327
C06597=1057.068,448.869,369.567,176.565,41.868,158.323
C06598=1057.050,448.624,369.613,176.551,41.857,158.318
C06599=1057.033,448.380,369.661,176.537,41.845,158.314
C06600=1057.017,448.136,369.709,176.523,41.833,158.310
C06601=1057.000,447.891,369.758,176.509,41.821,158.306
C06602=1056.986,447.646,369.808,176.495,41.809,158.302
C06603=1056.971,447.403,369.857,176.482,41.797,158.297
C06604=1056.958,447.160,369.908,176.468,41.784,158.293
C06605=1056.946,446.916,369.959,176.454,41.771,158.289
C06606=1056.934,446.673,370.010,176.441,41.758,158.284
C06607=1056.924,446.429,370.062,176.428,41.745,158.280
C06608=1056.912,446.185,370.114,176.414,41.732,158.275
C06609=1056.903,445.977,370.158,176.403,41.721,158.271
C06610=1056.892,445.769,370.203,176.392,41.710,158.268
C06611=1056.883,445.561,370.247,176.381,41.699,158.264
C06612=1056.873,445.352,370.290,176.370,41.688,158.260
C06613=1056.864,445.144,370.334,176.358,41.677,158.257
C06614=1056.854,444.936,370.378,176.348,41.666,158.253
C06615=1056.845,444.728,370.423,176.336,41.655,158.249
C06616=1056.835,444.519,370.466,176.325,41.644,158.245
C06617=1056.824,444.275,370.518,176.312,41.632,158.241
C06618=1056.813,444.031,370.569,176.300,41.619,158.237
C06619=1056.802,443.787,370.620,176.287,41.606,158.233
C06620=1056.791,443.541,370.671,176.274,41.593,158.228
C06621=1056.780,443.298,370.722,176.262,41.581,158.224
C06622=1056.769,443.053,370.774,176.249,41.568,158.220
C06623=1056.758,442.808,370.825,176.236,41.556,158.216
C06624=1056.747,442.564,370.876,176.224,41.543,158.212
C06625=1056.736,442.320,370.927,176.211,41.531,158.207
C06626=1056.725,442.075,370.979,176.199,41.518,158.203
C06627=1056.714,441.831,371.029,176.187,41.506,158.199
C06628=1056.703,441.586,371.079,176.174,41.494,158.195
C06629=1056.693,441.341,371.130,176.162,41.482,158.191
C06630=1056.681,441.098,371.181,176.150,41.470,158.187
C06631=1056.671,440.853,371.232,176.138,41.457,158.183
C06632=1056.660,440.608,371.283,176.126,41.445,158.179
C06633=1056.649,440.364,371.333,176.114,41.433,158.175
C06634=1056.639,440.119,371.384,176.102,41.421,158.171
C06635=1056.628,439.875,371.434,176.089,41.409,158.167
C06636=1056.617,439.630,371.485,176.078,41.397,158.163
C06637=1056.607,439.385,371.535,176.066,41.385,158.159
C06638=1056.596,439.141,371.585,176.054,41.373,158.155
C06639=1056.585,438.896,371.635,176.042,41.361,158.151
C06640=1056.574,438.651,371.685,176.031,41.349,158.147
C06641=1056.564,438.406,371.736,176.019,41.337,158.143
C06642=1056.554,438.161,371.785,176.008,41.326,158.140
C06643=1056.543,437.917,371.836,175.995,41.314,158.136
C06644=1056.532,437.672,371.885,175.984,41.302,158.132
C06645=1056.522,437.428,371.935,175.972,41.290,158.128
C06646=1056.512,437.183,371.986,175.961,41.279,158.124
C06647=1056.501,436.938,372.035,175.950,41.267,158.120
C06648=1056.490,436.693,372.085,175.939,41.256,158.117
C06649=1056.480,436.448,372.134,175.927,41.244,158.113
C06650=1056.470,436.203,372.184,175.916,41.233,158.109
C06651=1056.459,435.958,372.233,175.905,41.221,158.106
C06652=1056.449,435.714,372.283,175.894,41.210,158.102
C06653=1056.438,435.469,372.332,175.882,41.199,158.098
C06654=1056.428,435.224,372.382,175.871,41.187,158.094
C06655=1056.417,434.979,372.431,175.860,41.176,158.091
C06656=1056.407,434.734,372.481,175.849,41.165,158.087
C06657=1056.397,434.490,372.530,175.838,41.154,158.084
C06658=1056.386,434.244,372.579,175.827,41.142,158.080
C06659=1056.376,434.000,372.628,175.816,41.131,158.076
C06660=1056.366,433.754,372.677,175.806,41.120,158.073
C06661=1056.356,433.510,372.726,175.795,41.109,158.069
C06662=1056.345,433.265,372.774,175.783,41.098,158.066
C06663=1056.335,433.020,372.824,175.772,41.087,158.062
C06664=1056.325,432.775,372.872,175.762,41.076,158.059
C06665=1056.314,432.530,372.922,175.752,41.065,158.055
C06666=1056.304,432.285,372.970,175.741,41.054,158.052
C06667=1056.295,432.040,373.019,175.730,41.043,158.048
C06668=1056.285,431.795,373.067,175.720,41.032,158.045
C06669=1056.270,431.421,373.142,175.704,41.016,158.039
C06670=1056.254,431.046,373.216,175.688,40.999,158.034
C06671=1056.239,430.672,373.291,175.671,40.983,158.029
C06672=1056.224,430.297,373.365,175.656,40.966,158.024
C06673=1056.214,430.052,373.414,175.645,40.955,158.020
C06674=1056.204,429.807,373.461,175.635,40.945,158.017
C06675=1056.194,429.562,373.510,175.625,40.934,158.014
C06676=1056.184,429.317,373.558,175.614,40.924,158.010
C06677=1056.174,429.071,373.606,175.605,40.913,158.007
C06678=1056.164,428.826,373.654,175.595,40.903,158.004
C06679=1056.154,428.581,373.703,175.584,40.892,158.000
C06680=1056.144,428.336,373.750,175.575,40.882,157.997
C06681=1056.134,428.091,373.798,175.564,40.872,157.994
C06682=1056.125,427.845,373.846,175.554,40.861,157.991
C06683=1056.115,427.601,373.893,175.545,40.851,157.987
C06684=1056.105,427.356,373.942,175.534,40.841,157.984
C06685=1056.096,427.110,373.989,175.525,40.830,157.981
C06686=1056.086,426.865,374.037,175.515,40.820,157.978
C06687=1056.076,426.620,374.085,175.505,40.810,157.975
C06688=1056.066,426.374,374.133,175.495,40.799,157.971
C06689=1056.051,425.978,374.209,175.480,40.783,157.966
C06690=1056.035,425.584,374.286,175.464,40.767,157.961
C06691=1056.019,425.188,374.362,175.449,40.751,157.956
C06692=1056.004,424.792,374.439,175.433,40.735,157.951
C06693=1055.994,424.547,374.485,175.424,40.725,157.948
C06694=1055.985,424.301,374.533,175.414,40.715,157.945
C06695=1055.975,424.056,374.580,175.405,40.705,157.942
C06696=1055.965,423.811,374.627,175.396,40.695,157.939
C06697=1055.956,423.566,374.674,175.386,40.685,157.936
C06698=1055.946,423.320,374.721,175.377,40.675,157.933
C06699=1055.937,423.075,374.768,175.367,40.666,157.930
C06700=1055.927,422.829,374.815,175.358,40.656,157.927
C06701=1055.917,422.584,374.862,175.348,40.647,157.924
C06702=1055.908,422.338,374.909,175.339,40.636,157.921
C06703=1055.899,422.094,374.956,175.330,40.627,157.918
C06704=1055.889,421.848,375.002,175.322,40.617,157.915
C06705=1055.880,421.602,375.049,175.312,40.607,157.912
C06706=1055.870,421.357,375.096,175.303,40.598,157.909
C06707=1055.861,421.112,375.142,175.294,40.589,157.906
C06708=1055.852,420.866,375.189,175.285,40.579,157.903
C06709=1055.842,420.620,375.235,175.276,40.569,157.900
C06710=1055.833,420.375,375.282,175.267,40.560,157.898
C06711=1055.825,420.130,375.328,175.258,40.551,157.895
C06712=1055.815,419.884,375.375,175.248,40.541,157.892
C06713=1055.805,419.638,375.421,175.240,40.532,157.889
C06714=1055.796,419.393,375.467,175.231,40.522,157.886
C06715=1055.787,419.147,375.514,175.222,40.513,157.883
C06716=1055.778,418.902,375.560,175.213,40.504,157.881
C06717=1055.768,418.656,375.607,175.204,40.494,157.878
C06718=1055.759,418.410,375.652,175.196,40.485,157.875
C06719=1055.750,418.165,375.698,175.187,40.476,157.872
C06720=1055.740,417.920,375.745,175.178,40.467,157.869
C06721=1055.731,417.696,375.786,175.170,40.459,157.867
C06722=1055.723,417.471,375.829,175.163,40.450,157.864
C06723=1055.715,417.248,375.870,175.155,40.442,157.862
C06724=1055.706,417.024,375.912,175.146,40.434,157.859
C06725=1055.698,416.800,375.954,175.139,40.425,157.857
C06726=1055.690,416.577,375.995,175.131,40.417,157.854
C06727=1055.682,416.352,376.037,175.124,40.409,157.852
C06728=1055.673,416.128,376.079,175.116,40.400,157.849
C06729=1055.664,415.882,376.125,175.107,40.392,157.847
C06730=1055.655,415.637,376.171,175.099,40.382,157.844
C06731=1055.646,415.391,376.216,175.090,40.374,157.841
C06732=1055.637,415.146,376.262,175.082,40.364,157.839
C06733=1055.628,414.900,376.307,175.074,40.356,157.836
C06734=1055.619,414.654,376.352,175.065,40.347,157.833
C06735=1055.610,414.409,376.399,175.057,40.338,157.831
C06736=1055.601,414.164,376.444,175.048,40.329,157.828
C06737=1055.592,413.918,376.489,175.040,40.320,157.825
C06738=1055.583,413.672,376.534,175.032,40.312,157.823
C06739=1055.574,413.426,376.580,175.024,40.303,157.820
C06740=1055.565,413.180,376.625,175.016,40.294,157.818
C06741=1055.556,412.934,376.669,175.007,40.285,157.815
C06742=1055.547,412.688,376.715,175.000,40.277,157.812
C06743=1055.538,412.443,376.760,174.991,40.269,157.810
C06744=1055.528,412.197,376.805,174.983,40.260,157.807
C06745=1055.520,411.952,376.850,174.975,40.251,157.805
C06746=1055.511,411.705,376.895,174.967,40.243,157.802
C06747=1055.502,411.460,376.940,174.959,40.234,157.800
C06748=1055.493,411.213,376.984,174.951,40.226,157.797
C06749=1055.484,410.968,377.029,174.943,40.217,157.795
C06750=1055.475,410.723,377.075,174.936,40.209,157.792
C06751=1055.466,410.476,377.119,174.927,40.200,157.790
C06752=1055.457,410.231,377.164,174.919,40.192,157.787
C06753=1055.449,409.985,377.209,174.912,40.183,157.785
C06754=1055.440,409.739,377.253,174.903,40.175,157.782
C06755=1055.431,409.494,377.298,174.896,40.167,157.780
C06756=1055.422,409.247,377.342,174.888,40.158,157.777
C06757=1055.413,409.001,377.387,174.880,40.150,157.775
C06758=1055.405,408.756,377.432,174.872,40.142,157.772
C06759=1055.395,408.510,377.476,174.864,40.133,157.770
C06760=1055.387,408.264,377.520,174.857,40.125,157.768
C06761=1055.379,408.018,377.565,174.849,40.117,157.765
C06762=1055.370,407.772,377.609,174.842,40.109,157.763
C06763=1055.361,407.526,377.653,174.834,40.101,157.761
C06764=1055.353,407.281,377.698,174.826,40.093,157.758
C06765=1055.343,407.034,377.742,174.819,40.084,157.756
C06766=1055.335,406.789,377.787,174.811,40.076,157.753
C06767=1055.326,406.543,377.830,174.804,40.068,157.751
C06768=1055.318,406.296,377.874,174.796,40.060,157.749
C06769=1055.309,406.051,377.918,174.789,40.052,157.746
C06770=1055.301,405.805,377.963,174.780,40.044,157.744
C06771=1055.293,405.559,378.007,174.773,40.036,157.742
C06772=1055.284,405.313,378.051,174.766,40.028,157.739
C06773=1055.276,405.067,378.095,174.758,40.020,157.737
C06774=1055.267,404.821,378.139,174.751,40.012,157.735
C06775=1055.258,404.575,378.183,174.744,40.004,157.732
C06776=1055.250,404.329,378.227,174.736,39.996,157.730
C06777=1055.241,404.083,378.270,174.729,39.988,157.728
C06778=1055.233,403.837,378.315,174.722,39.980,157.726
C06779=1055.224,403.591,378.358,174.714,39.973,157.723
C06780=1055.216,403.345,378.402,174.707,39.965,157.721
C06781=1055.204,402.998,378.463,174.697,39.954,157.718
C06782=1055.192,402.652,378.524,174.686,39.943,157.715
C06783=1055.179,402.305,378.586,174.676,39.932,157.712
C06784=1055.168,401.958,378.647,174.666,39.921,157.708
C06785=1055.159,401.712,378.690,174.659,39.914,157.706
C06786=1055.151,401.466,378.734,174.652,39.906,157.704
C06787=1055.142,401.219,378.777,174.644,39.898,157.702
C06788=1055.133,400.974,378.821,174.638,39.891,157.700
C06789=1055.125,400.728,378.864,174.631,39.883,157.697
C06790=1055.116,400.482,378.907,174.624,39.876,157.695
C06791=1055.108,400.235,378.950,174.617,39.868,157.693
C06792=1055.100,399.989,378.994,174.609,39.860,157.691
C06793=1055.092,399.743,379.037,174.602,39.853,157.689
C06794=1055.083,399.497,379.080,174.595,39.845,157.687
C06795=1055.075,399.251,379.123,174.589,39.838,157.685
C06796=1055.066,399.005,379.166,174.582,39.831,157.683
C06797=1055.058,398.759,379.209,174.575,39.823,157.680
C06798=1055.050,398.513,379.251,174.568,39.816,157.678
C06799=1055.042,398.267,379.294,174.561,39.809,157.676
C06800=1055.034,398.020,379.337,174.554,39.801,157.674
C06801=1055.025,397.774,379.380,174.547,39.793,157.672
C06802=1055.017,397.528,379.423,174.540,39.786,157.670
C06803=1055.009,397.282,379.466,174.533,39.779,157.668
C06804=1055.001,397.036,379.508,174.527,39.771,157.666
C06805=1054.992,396.790,379.551,174.520,39.765,157.664
C06806=1054.984,396.544,379.594,174.513,39.757,157.662
C06807=1054.975,396.298,379.637,174.506,39.750,157.660
C06808=1054.967,396.051,379.679,174.500,39.743,157.658
C06809=1054.959,395.805,379.722,174.493,39.736,157.656
C06810=1054.950,395.559,379.763,174.486,39.728,157.653
C06811=1054.942,395.313,379.806,174.479,39.721,157.651
C06812=1054.934,395.066,379.849,174.473,39.714,157.649
C06813=1054.926,394.821,379.891,174.466,39.707,157.647
C06814=1054.918,394.574,379.934,174.459,39.700,157.645
C06815=1054.909,394.328,379.976,174.453,39.693,157.643
C06816=1054.902,394.082,380.019,174.446,39.686,157.641
C06817=1054.893,393.836,380.061,174.439,39.679,157.639
C06818=1054.885,393.590,380.102,174.433,39.672,157.637
C06819=1054.877,393.343,380.145,174.426,39.665,157.636
C06820=1054.869,393.097,380.187,174.420,39.657,157.633
C06821=1054.861,392.851,380.230,174.413,39.651,157.632
C06822=1054.853,392.605,380.272,174.406,39.644,157.630
C06823=1054.845,392.359,380.314,174.400,39.637,157.628
C06824=1054.836,392.112,380.356,174.393,39.630,157.626
C06825=1054.828,391.866,380.398,174.387,39.623,157.624
C06826=1054.820,391.620,380.440,174.380,39.616,157.622
C06827=1054.812,391.374,380.481,174.374,39.609,157.620
C06828=1054.804,391.127,380.523,174.368,39.602,157.618
C06829=1054.796,390.881,380.565,174.361,39.595,157.616
C06830=1054.787,390.634,380.606,174.355,39.589,157.614
C06831=1054.780,390.388,380.648,174.348,39.582,157.612
C06832=1054.772,390.142,380.690,174.342,39.575,157.610
C06833=1054.763,389.896,380.732,174.335,39.568,157.609
C06834=1054.756,389.650,380.774,174.329,39.561,157.607
C06835=1054.748,389.403,380.816,174.323,39.555,157.605
C06836=1054.740,389.157,380.857,174.317,39.548,157.603
C06837=1054.729,388.828,380.912,174.308,39.539,157.600
C06838=1054.718,388.499,380.968,174.300,39.530,157.598
C06839=1054.707,388.170,381.022,174.292,39.522,157.596
C06840=1054.697,387.842,381.078,174.283,39.513,157.593
C06841=1054.689,387.594,381.120,174.276,39.506,157.591
C06842=1054.680,387.349,381.161,174.271,39.500,157.589
C06843=1054.672,387.103,381.202,174.265,39.493,157.588
C06844=1054.664,386.856,381.244,174.258,39.486,157.586
C06845=1054.656,386.610,381.284,174.252,39.480,157.584
C06846=1054.649,386.363,381.326,174.246,39.474,157.582
C06847=1054.640,386.117,381.367,174.240,39.467,157.580
C06848=1054.632,385.870,381.408,174.234,39.460,157.579
C06849=1054.625,385.624,381.449,174.227,39.454,157.577
C06850=1054.617,385.377,381.490,174.222,39.448,157.575
C06851=1054.609,385.131,381.532,174.215,39.441,157.573
C06852=1054.601,384.885,381.573,174.209,39.435,157.572
C06853=1054.593,384.639,381.613,174.204,39.428,157.570
C06854=1054.585,384.392,381.655,174.197,39.422,157.568
C06855=1054.577,384.145,381.695,174.191,39.415,157.566
C06856=1054.570,383.899,381.737,174.185,39.409,157.564
C06857=1054.562,383.652,381.777,174.179,39.402,157.563
C06858=1054.554,383.406,381.818,174.173,39.397,157.561
C06859=1054.546,383.160,381.859,174.167,39.390,157.559
C06860=1054.538,382.913,381.900,174.162,39.384,157.557
C06861=1054.530,382.667,381.940,174.155,39.377,157.556
C06862=1054.523,382.420,381.982,174.149,39.371,157.554
C06863=1054.515,382.174,382.022,174.144,39.365,157.552
C06864=1054.507,381.928,382.063,174.137,39.358,157.550
C06865=1054.500,381.681,382.103,174.132,39.352,157.549
C06866=1054.492,381.434,382.144,174.126,39.346,157.547
C06867=1054.484,381.188,382.185,174.120,39.339,157.545
C06868=1054.477,380.941,382.226,174.114,39.334,157.544
C06869=1054.469,380.695,382.266,174.108,39.327,157.542
C06870=1054.461,380.448,382.306,174.102,39.321,157.540
C06871=1054.454,380.202,382.348,174.097,39.315,157.539
C06872=1054.446,379.955,382.388,174.091,39.309,157.537
C06873=1054.438,379.708,382.428,174.085,39.303,157.535
C06874=1054.430,379.462,382.468,174.079,39.296,157.534
C06875=1054.422,379.215,382.509,174.073,39.290,157.532
C06876=1054.415,378.969,382.548,174.068,39.285,157.530
C06877=1054.407,378.723,382.589,174.062,39.278,157.529
C06878=1054.399,378.476,382.629,174.056,39.272,157.527
C06879=1054.391,378.229,382.669,174.050,39.266,157.525
C06880=1054.383,377.983,382.709,174.045,39.260,157.524
C06881=1054.376,377.736,382.749,174.039,39.255,157.522
C06882=1054.368,377.489,382.789,174.034,39.248,157.521
C06883=1054.361,377.243,382.830,174.028,39.242,157.519
C06884=1054.353,376.996,382.869,174.022,39.236,157.517
C06885=1054.345,376.750,382.909,174.016,39.231,157.516
C06886=1054.337,376.503,382.949,174.011,39.225,157.514
C06887=1054.329,376.256,382.990,174.005,39.219,157.513
C06888=1054.322,376.010,383.029,174.000,39.213,157.511
C06889=1054.315,375.763,383.069,173.994,39.207,157.509
C06890=1054.307,375.516,383.109,173.989,39.201,157.508
C06891=1054.299,375.269,383.149,173.983,39.195,157.506
C06892=1054.292,375.023,383.189,173.978,39.189,157.505
C06893=1054.282,374.726,383.237,173.971,39.182,157.503
C06894=1054.273,374.429,383.285,173.964,39.175,157.501
C06895=1054.264,374.133,383.332,173.957,39.168,157.499
C06896=1054.255,373.835,383.381,173.951,39.161,157.497
C06897=1054.248,373.589,383.420,173.945,39.155,157.496
C06898=1054.240,373.342,383.460,173.940,39.150,157.494
C06899=1054.233,373.095,383.500,173.934,39.144,157.492
C06900=1054.226,372.848,383.539,173.929,39.138,157.491
C06901=1054.218,372.601,383.579,173.923,39.132,157.489
C06902=1054.210,372.355,383.618,173.918,39.126,157.488
C06903=1054.203,372.109,383.658,173.912,39.120,157.486
C06904=1054.195,371.862,383.697,173.907,39.115,157.485
C06905=1054.188,371.615,383.736,173.902,39.109,157.483
C06906=1054.180,371.368,383.776,173.896,39.104,157.482
C06907=1054.173,371.121,383.814,173.891,39.098,157.480
C06908=1054.165,370.875,383.854,173.885,39.093,157.479
C06909=1054.158,370.628,383.893,173.880,39.087,157.477
C06910=1054.150,370.381,383.933,173.875,39.081,157.476
C06911=1054.143,370.134,383.971,173.869,39.076,157.474
C06912=1054.135,369.887,384.011,173.864,39.070,157.473
C06913=1054.128,369.641,384.050,173.858,39.065,157.471
C06914=1054.120,369.394,384.089,173.853,39.059,157.470
C06915=1054.112,369.147,384.128,173.848,39.054,157.468
C06916=1054.105,368.901,384.168,173.842,39.048,157.467
C06917=1054.098,368.654,384.206,173.838,39.042,157.465
C06918=1054.090,368.406,384.245,173.833,39.037,157.464
C06919=1054.083,368.160,384.285,173.827,39.032,157.462
C06920=1054.074,367.913,384.323,173.822,39.026,157.461
C06921=1054.068,367.666,384.362,173.817,39.021,157.460
C06922=1054.061,367.419,384.401,173.811,39.015,157.458
C06923=1054.052,367.173,384.440,173.806,39.009,157.457
C06924=1054.046,366.926,384.479,173.801,39.004,157.455
C06925=1054.037,366.679,384.518,173.795,38.999,157.454
C06926=1054.031,366.432,384.557,173.791,38.993,157.452
C06927=1054.024,366.185,384.595,173.786,38.988,157.451
C06928=1054.016,365.939,384.634,173.780,38.982,157.449
C06929=1054.009,365.692,384.674,173.775,38.977,157.448
C06930=1054.001,365.445,384.712,173.770,38.972,157.447
C06931=1053.994,365.198,384.751,173.764,38.966,157.445
C06932=1053.986,364.951,384.789,173.759,38.961,157.444
C06933=1053.979,364.704,384.828,173.755,38.955,157.442
C06934=1053.972,364.458,384.866,173.750,38.950,157.441
C06935=1053.965,364.211,384.905,173.744,38.945,157.440
C06936=1053.957,363.963,384.944,173.739,38.940,157.438
C06937=1053.950,363.716,384.982,173.734,38.934,157.437
C06938=1053.943,363.470,385.021,173.730,38.929,157.435
C06939=1053.936,363.223,385.059,173.724,38.923,157.434
C06940=1053.928,362.977,385.097,173.719,38.919,157.433
C06941=1053.921,362.729,385.136,173.714,38.913,157.431
C06942=1053.914,362.482,385.174,173.709,38.908,157.430
C06943=1053.906,362.235,385.212,173.704,38.903,157.428
C06944=1053.899,361.988,385.251,173.699,38.897,157.427
C06945=1053.892,361.741,385.289,173.694,38.893,157.426
C06946=1053.884,361.494,385.327,173.689,38.887,157.424
C06947=1053.876,361.248,385.365,173.684,38.882,157.423
C06948=1053.870,361.000,385.404,173.679,38.877,157.422
C06949=1053.861,360.722,385.447,173.674,38.871,157.420
C06950=1053.853,360.445,385.489,173.668,38.865,157.419
C06951=1053.845,360.166,385.532,173.662,38.859,157.417
C06952=1053.836,359.887,385.575,173.657,38.853,157.416
C06953=1053.829,359.640,385.613,173.651,38.849,157.414
C06954=1053.822,359.394,385.651,173.647,38.844,157.413
C06955=1053.814,359.147,385.689,173.642,38.838,157.412
C06956=1053.808,358.900,385.728,173.637,38.833,157.410
C06957=1053.800,358.653,385.765,173.633,38.828,157.409
C06958=1053.793,358.406,385.803,173.627,38.823,157.408
C06959=1053.786,358.159,385.841,173.622,38.818,157.406
C06960=1053.779,357.912,385.879,173.618,38.813,157.405
C06961=1053.772,357.664,385.917,173.613,38.808,157.404
C06962=1053.764,357.418,385.955,173.608,38.803,157.402
C06963=1053.757,357.171,385.992,173.604,38.798,157.401
C06964=1053.750,356.924,386.030,173.598,38.793,157.400
C06965=1053.743,356.677,386.067,173.593,38.788,157.398
C06966=1053.735,356.429,386.105,173.589,38.783,157.397
C06967=1053.728,356.182,386.142,173.584,38.778,157.396
C06968=1053.721,355.936,386.181,173.579,38.773,157.395
C06969=1053.713,355.689,386.218,173.575,38.768,157.393
C06970=1053.706,355.441,386.256,173.570,38.764,157.392
C06971=1053.699,355.194,386.293,173.565,38.759,157.391
C06972=1053.692,354.947,386.331,173.560,38.754,157.390
C06973=1053.684,354.700,386.368,173.555,38.749,157.388
C06974=1053.677,354.453,386.406,173.551,38.744,157.387
C06975=1053.670,354.207,386.443,173.546,38.739,157.386
C06976=1053.663,353.959,386.480,173.541,38.734,157.384
C06977=1053.656,353.712,386.518,173.537,38.729,157.383
C06978=1053.649,353.464,386.555,173.532,38.724,157.382
C06979=1053.642,353.217,386.592,173.528,38.719,157.381
C06980=1053.635,352.970,386.630,173.522,38.714,157.379
C06981=1053.627,352.723,386.667,173.518,38.709,157.378
C06982=1053.621,352.477,386.705,173.513,38.704,157.377
C06983=1053.613,352.230,386.742,173.508,38.700,157.376
C06984=1053.606,351.982,386.779,173.504,38.695,157.374
C06985=1053.599,351.735,386.816,173.499,38.690,157.373
C06986=1053.592,351.487,386.854,173.495,38.685,157.372
C06987=1053.585,351.241,386.891,173.490,38.680,157.371
C06988=1053.578,350.993,386.928,173.486,38.676,157.370
C06989=1053.570,350.746,386.965,173.481,38.671,157.368
C06990=1053.563,350.499,387.002,173.476,38.666,157.367
C06991=1053.557,350.252,387.039,173.471,38.662,157.366
C06992=1053.550,350.005,387.076,173.467,38.657,157.365
C06993=1053.542,349.758,387.113,173.462,38.652,157.364
C06994=1053.535,349.511,387.150,173.458,38.648,157.362
C06995=1053.528,349.264,387.187,173.453,38.643,157.361
C06996=1053.521,349.016,387.224,173.449,38.638,157.360
C06997=1053.513,348.769,387.260,173.444,38.633,157.359
C06998=1053.507,348.522,387.297,173.440,38.629,157.357
C06999=1053.500,348.275,387.334,173.435,38.624,157.356
C07000=1053.493,348.027,387.371,173.431,38.620,157.355
C07001=1053.485,347.781,387.408,173.426,38.615,157.354
C07002=1053.479,347.533,387.444,173.422,38.610,157.353
C07003=1053.472,347.285,387.481,173.417,38.605,157.351
C07004=1053.464,347.039,387.518,173.413,38.601,157.350
C07005=1053.457,346.766,387.559,173.408,38.596,157.349
C07006=1053.449,346.493,387.599,173.403,38.590,157.348
C07007=1053.441,346.220,387.640,173.397,38.586,157.346
C07008=1053.433,345.946,387.680,173.393,38.581,157.345
C07009=1053.426,345.699,387.717,173.388,38.576,157.344
C07010=1053.419,345.452,387.753,173.384,38.571,157.343
C07011=1053.412,345.204,387.790,173.379,38.567,157.342
C07012=1053.405,344.957,387.826,173.375,38.562,157.341
C07013=1053.398,344.710,387.863,173.371,38.557,157.339
C07014=1053.391,344.463,387.898,173.366,38.553,157.338
C07015=1053.384,344.216,387.936,173.362,38.549,157.337
C07016=1053.378,343.969,387.972,173.357,38.544,157.336
C07017=1053.370,343.721,388.009,173.353,38.539,157.335
C07018=1053.364,343.474,388.045,173.349,38.535,157.334
C07019=1053.356,343.227,388.081,173.344,38.530,157.332
C07020=1053.350,342.980,388.118,173.340,38.526,157.331
C07021=1053.342,342.732,388.154,173.336,38.522,157.330
C07022=1053.336,342.484,388.190,173.331,38.517,157.329
C07023=1053.328,342.237,388.226,173.327,38.513,157.328
C07024=1053.322,341.990,388.262,173.323,38.508,157.327
C07025=1053.314,341.743,388.299,173.318,38.503,157.326
C07026=1053.307,341.496,388.334,173.314,38.499,157.324
C07027=1053.300,341.248,388.371,173.310,38.495,157.323
C07028=1053.294,341.001,388.406,173.306,38.490,157.322
C07029=1053.286,340.753,388.443,173.302,38.486,157.321
C07030=1053.280,340.506,388.479,173.297,38.481,157.320
C07031=1053.272,340.259,388.515,173.293,38.477,157.319
C07032=1053.266,340.011,388.551,173.289,38.473,157.318
C07033=1053.259,339.764,388.587,173.284,38.469,157.317
C07034=1053.251,339.517,388.623,173.280,38.464,157.316
C07035=1053.245,339.269,388.659,173.276,38.460,157.315
C07036=1053.238,339.022,388.695,173.271,38.455,157.313
C07037=1053.230,338.775,388.731,173.267,38.451,157.312
C07038=1053.224,338.527,388.767,173.263,38.446,157.311
C07039=1053.217,338.281,388.802,173.259,38.442,157.310
C07040=1053.210,338.032,388.838,173.254,38.438,157.309
C07041=1053.204,337.785,388.874,173.250,38.434,157.308
C07042=1053.197,337.538,388.909,173.246,38.429,157.307
C07043=1053.190,337.291,388.945,173.243,38.425,157.306
C07044=1053.183,337.043,388.981,173.238,38.420,157.305
C07045=1053.176,336.796,389.017,173.234,38.416,157.304
C07046=1053.169,336.549,389.052,173.230,38.412,157.303
C07047=1053.162,336.301,389.089,173.226,38.408,157.302
C07048=1053.155,336.054,389.124,173.221,38.403,157.300
C07049=1053.149,335.806,389.159,173.217,38.399,157.299
C07050=1053.142,335.560,389.195,173.213,38.395,157.298
C07051=1053.134,335.312,389.231,173.209,38.391,157.297
C07052=1053.128,335.064,389.266,173.204,38.386,157.296
C07053=1053.121,334.817,389.301,173.200,38.382,157.295
C07054=1053.114,334.570,389.337,173.197,38.378,157.294
C07055=1053.106,334.322,389.372,173.193,38.374,157.293
C07056=1053.100,334.075,389.408,173.188,38.369,157.292
C07057=1053.093,333.827,389.443,173.184,38.365,157.291
C07058=1053.086,333.580,389.478,173.180,38.361,157.290
C07059=1053.079,333.333,389.514,173.176,38.357,157.289
C07060=1053.072,333.085,389.550,173.172,38.353,157.288
C07061=1053.064,332.808,389.589,173.167,38.348,157.287
C07062=1053.057,332.531,389.628,173.162,38.343,157.286
C07063=1053.049,332.253,389.668,173.158,38.339,157.284
C07064=1053.042,331.977,389.708,173.153,38.334,157.283
C07065=1053.035,331.729,389.743,173.150,38.330,157.282
C07066=1053.028,331.482,389.778,173.146,38.326,157.281
C07067=1053.021,331.235,389.813,173.142,38.322,157.280
C07068=1053.014,330.987,389.848,173.138,38.317,157.279
C07069=1053.007,330.739,389.884,173.134,38.313,157.278
C07070=1053.000,330.492,389.919,173.129,38.309,157.277
C07071=1052.994,330.244,389.953,173.125,38.305,157.276
C07072=1052.987,329.996,389.988,173.121,38.301,157.275
C07073=1052.980,329.749,390.023,173.118,38.297,157.274
C07074=1052.974,329.502,390.059,173.114,38.293,157.273
C07075=1052.966,329.255,390.093,173.110,38.289,157.272
C07076=1052.959,329.007,390.128,173.105,38.284,157.271
C07077=1052.953,328.759,390.163,173.101,38.280,157.270
C07078=1052.945,328.512,390.197,173.097,38.277,157.269
C07079=1052.938,328.264,390.233,173.094,38.273,157.268
C07080=1052.931,328.016,390.267,173.090,38.269,157.267
C07081=1052.924,327.769,390.302,173.086,38.265,157.266
C07082=1052.917,327.522,390.337,173.082,38.260,157.265
C07083=1052.911,327.274,390.371,173.078,38.256,157.264
C07084=1052.903,327.027,390.406,173.074,38.253,157.263
C07085=1052.896,326.779,390.441,173.070,38.249,157.262
C07086=1052.890,326.531,390.475,173.066,38.245,157.261
C07087=1052.883,326.284,390.510,173.062,38.241,157.260
C07088=1052.876,326.036,390.544,173.058,38.237,157.259
C07089=1052.869,325.789,390.579,173.054,38.233,157.258
C07090=1052.862,325.541,390.613,173.051,38.229,157.257
C07091=1052.855,325.294,390.648,173.047,38.225,157.256
C07092=1052.848,325.046,390.682,173.043,38.221,157.255
C07093=1052.841,324.799,390.717,173.039,38.217,157.254
C07094=1052.835,324.552,390.751,173.035,38.213,157.253
C07095=1052.828,324.305,390.786,173.031,38.209,157.252
C07096=1052.822,324.057,390.820,173.027,38.205,157.251
C07097=1052.814,323.810,390.855,173.023,38.201,157.250
C07098=1052.808,323.562,390.889,173.019,38.197,157.249
C07099=1052.801,323.314,390.924,173.016,38.193,157.249
C07100=1052.794,323.066,390.958,173.012,38.190,157.248
C07101=1052.787,322.819,390.993,173.008,38.186,157.247
C07102=1052.781,322.572,391.026,173.004,38.182,157.246
C07103=1052.774,322.324,391.061,173.000,38.178,157.245
C07104=1052.767,322.076,391.096,172.997,38.174,157.244
C07105=1052.760,321.829,391.130,172.993,38.170,157.243
C07106=1052.753,321.581,391.165,172.989,38.166,157.242
C07107=1052.747,321.334,391.198,172.985,38.162,157.241
C07108=1052.740,321.086,391.233,172.981,38.158,157.240
C07109=1052.733,320.839,391.266,172.978,38.154,157.239
C07110=1052.726,320.591,391.301,172.974,38.150,157.238
C07111=1052.720,320.343,391.336,172.970,38.146,157.237
C07112=1052.713,320.096,391.369,172.966,38.142,157.236
C07113=1052.707,319.848,391.404,172.963,38.138,157.235
C07114=1052.700,319.601,391.438,172.959,38.135,157.234
C07115=1052.694,319.353,391.472,172.955,38.131,157.233
C07116=1052.686,319.106,391.505,172.951,38.127,157.232
C07117=1052.679,318.823,391.545,172.947,38.123,157.231
C07118=1052.672,318.540,391.584,172.944,38.118,157.230
C07119=1052.663,318.258,391.622,172.939,38.114,157.229
C07120=1052.656,317.976,391.661,172.935,38.109,157.228
C07121=1052.650,317.728,391.696,172.931,38.105,157.227
C07122=1052.643,317.481,391.729,172.927,38.101,157.226
C07123=1052.637,317.233,391.764,172.924,38.098,157.225
C07124=1052.630,316.986,391.797,172.920,38.094,157.224
C07125=1052.624,316.738,391.831,172.916,38.090,157.223
C07126=1052.617,316.491,391.865,172.912,38.086,157.222
C07127=1052.610,316.243,391.900,172.908,38.082,157.221
C07128=1052.604,315.996,391.933,172.906,38.078,157.221
C07129=1052.597,315.748,391.968,172.902,38.075,157.220
C07130=1052.591,315.500,392.000,172.898,38.071,157.219
C07131=1052.584,315.252,392.035,172.895,38.067,157.218
C07132=1052.578,315.005,392.068,172.891,38.063,157.217
C07133=1052.571,314.757,392.103,172.887,38.059,157.216
C07134=1052.565,314.510,392.136,172.883,38.056,157.215
C07135=1052.558,314.262,392.170,172.880,38.052,157.214
C07136=1052.552,314.015,392.203,172.877,38.048,157.213
C07137=1052.545,313.767,392.237,172.873,38.044,157.212
C07138=1052.539,313.520,392.271,172.869,38.041,157.211
C07139=1052.532,313.272,392.305,172.866,38.037,157.210
C07140=1052.526,313.024,392.338,172.862,38.033,157.210
C07141=1052.519,312.776,392.372,172.858,38.029,157.209
C07142=1052.512,312.528,392.405,172.854,38.025,157.208
C07143=1052.505,312.281,392.438,172.851,38.022,157.207
C07144=1052.498,312.033,392.471,172.848,38.018,157.206
C07145=1052.491,311.786,392.505,172.844,38.015,157.205
C07146=1052.484,311.538,392.538,172.841,38.011,157.204
C07147=1052.478,311.291,392.571,172.837,38.007,157.203
C07148=1052.471,311.043,392.604,172.833,38.003,157.202
C07149=1052.464,310.795,392.638,172.830,38.000,157.202
C07150=1052.457,310.547,392.671,172.826,37.997,157.201
C07151=1052.450,310.300,392.705,172.822,37.993,157.200
C07152=1052.444,310.052,392.737,172.819,37.989,157.199
C07153=1052.437,309.804,392.771,172.816,37.985,157.198
C07154=1052.430,309.557,392.804,172.812,37.982,157.197
C07155=1052.424,309.309,392.837,172.808,37.978,157.196
C07156=1052.417,309.062,392.871,172.805,37.975,157.196
C07157=1052.410,308.814,392.903,172.801,37.971,157.195
C07158=1052.403,308.566,392.936,172.798,37.967,157.194
C07159=1052.396,308.319,392.969,172.795,37.964,157.193
C07160=1052.389,308.071,393.002,172.791,37.960,157.192
C07161=1052.383,307.823,393.035,172.787,37.956,157.191
C07162=1052.377,307.575,393.068,172.784,37.953,157.190
C07163=1052.370,307.328,393.102,172.780,37.949,157.190
C07164=1052.363,307.080,393.134,172.777,37.946,157.189
C07165=1052.356,306.832,393.168,172.774,37.942,157.188
C07166=1052.350,306.584,393.200,172.770,37.938,157.187
C07167=1052.343,306.338,393.233,172.766,37.935,157.186
C07168=1052.336,306.089,393.266,172.763,37.932,157.185
C07169=1052.330,305.842,393.299,172.760,37.928,157.184
C07170=1052.323,305.594,393.332,172.756,37.924,157.184
C07171=1052.316,305.346,393.365,172.752,37.920,157.183
C07172=1052.310,305.098,393.398,172.749,37.917,157.182
C07173=1052.303,304.820,393.434,172.745,37.913,157.181
C07174=1052.295,304.542,393.471,172.741,37.909,157.180
C07175=1052.288,304.264,393.509,172.738,37.905,157.179
C07176=1052.280,303.986,393.545,172.734,37.901,157.178
C07177=1052.274,303.738,393.578,172.730,37.897,157.177
C07178=1052.267,303.491,393.611,172.727,37.894,157.176
C07179=1052.260,303.243,393.643,172.724,37.890,157.176
C07180=1052.254,302.996,393.676,172.720,37.887,157.175
C07181=1052.247,302.748,393.709,172.716,37.883,157.174
C07182=1052.241,302.500,393.742,172.714,37.879,157.173
C07183=1052.235,302.252,393.774,172.710,37.876,157.172
C07184=1052.229,302.004,393.806,172.706,37.872,157.171
C07185=1052.221,301.756,393.839,172.703,37.869,157.170
C07186=1052.215,301.509,393.872,172.700,37.865,157.170
C07187=1052.208,301.261,393.904,172.697,37.862,157.169
C07188=1052.202,301.013,393.937,172.693,37.858,157.168
C07189=1052.196,300.766,393.970,172.690,37.854,157.167
C07190=1052.189,300.518,394.002,172.687,37.851,157.166
C07191=1052.182,300.270,394.035,172.683,37.847,157.165
C07192=1052.176,300.022,394.067,172.680,37.843,157.165
C07193=1052.170,299.774,394.100,172.677,37.840,157.164
C07194=1052.163,299.527,394.133,172.673,37.837,157.163
C07195=1052.156,299.280,394.165,172.670,37.833,157.162
C07196=1052.150,299.031,394.197,172.667,37.829,157.161
C07197=1052.144,298.784,394.230,172.663,37.826,157.160
C07198=1052.138,298.536,394.262,172.660,37.822,157.160
C07199=1052.132,298.289,394.295,172.657,37.818,157.159
C07200=1052.125,298.041,394.327,172.653,37.815,157.158
C07201=1052.118,297.793,394.359,172.650,37.812,157.157
C07202=1052.112,297.545,394.392,172.647,37.808,157.156
C07203=1052.106,297.297,394.424,172.644,37.805,157.155
C07204=1052.099,297.049,394.457,172.640,37.801,157.154
C07205=1052.093,296.801,394.489,172.637,37.797,157.154
C07206=1052.086,296.553,394.521,172.634,37.794,157.153
C07207=1052.080,296.306,394.554,172.631,37.790,157.152
C07208=1052.073,296.058,394.586,172.627,37.787,157.151
C07209=1052.067,295.810,394.618,172.624,37.784,157.150
C07210=1052.060,295.562,394.650,172.621,37.780,157.150
C07211=1052.054,295.314,394.682,172.618,37.777,157.149
C07212=1052.047,295.067,394.714,172.614,37.773,157.148
C07213=1052.041,294.819,394.746,172.611,37.769,157.147
C07214=1052.034,294.571,394.778,172.608,37.766,157.146
C07215=1052.028,294.323,394.810,172.604,37.762,157.146
C07216=1052.021,294.076,394.842,172.601,37.759,157.145
C07217=1052.014,293.828,394.874,172.598,37.756,157.144
C07218=1052.009,293.580,394.906,172.595,37.752,157.143
C07219=1052.001,293.333,394.938,172.592,37.749,157.142
C07220=1051.995,293.084,394.970,172.588,37.745,157.142
C07221=1051.989,292.836,395.001,172.585,37.742,157.141
C07222=1051.982,292.589,395.033,172.582,37.738,157.140
C07223=1051.976,292.341,395.065,172.579,37.735,157.139
C07224=1051.969,292.093,395.097,172.576,37.732,157.138
C07225=1051.962,291.845,395.128,172.572,37.729,157.138
C07226=1051.956,291.597,395.160,172.570,37.725,157.137
C07227=1051.949,291.350,395.193,172.566,37.722,157.136
C07228=1051.943,291.102,395.224,172.563,37.718,157.135
C07229=1051.936,290.839,395.257,172.560,37.714,157.134
C07230=1051.929,290.577,395.291,172.556,37.711,157.134
C07231=1051.922,290.315,395.325,172.553,37.708,157.133
C07232=1051.916,290.053,395.358,172.550,37.704,157.132
C07233=1051.909,289.805,395.389,172.546,37.701,157.131
C07234=1051.902,289.557,395.421,172.544,37.697,157.130
C07235=1051.896,289.309,395.453,172.540,37.694,157.130
C07236=1051.889,289.061,395.484,172.537,37.690,157.129
C07237=1051.883,288.813,395.516,172.534,37.687,157.128
C07238=1051.876,288.565,395.549,172.530,37.683,157.127
C07239=1051.870,288.317,395.580,172.528,37.680,157.126
C07240=1051.863,288.069,395.611,172.524,37.677,157.126
C07241=1051.857,287.822,395.642,172.522,37.673,157.125
C07242=1051.850,287.574,395.673,172.518,37.670,157.124
C07243=1051.844,287.326,395.705,172.516,37.667,157.123
C07244=1051.837,287.078,395.736,172.512,37.663,157.123
C07245=1051.831,286.830,395.768,172.509,37.660,157.122
C07246=1051.824,286.582,395.800,172.506,37.657,157.121
C07247=1051.817,286.334,395.831,172.503,37.653,157.120
C07248=1051.811,286.086,395.862,172.500,37.650,157.119
C07249=1051.804,285.838,395.894,172.497,37.647,157.119
C07250=1051.798,285.590,395.924,172.493,37.643,157.118
C07251=1051.791,285.342,395.956,172.491,37.640,157.117
C07252=1051.785,285.095,395.987,172.487,37.637,157.116
C07253=1051.778,284.847,396.018,172.485,37.634,157.116
C07254=1051.771,284.599,396.050,172.481,37.630,157.115
C07255=1051.765,284.350,396.081,172.479,37.627,157.114
C07256=1051.759,284.103,396.112,172.475,37.623,157.113
C07257=1051.752,283.855,396.143,172.472,37.620,157.113
C07258=1051.746,283.607,396.174,172.469,37.617,157.112
C07259=1051.739,283.359,396.205,172.466,37.613,157.111
C07260=1051.733,283.111,396.236,172.463,37.610,157.110
C07261=1051.726,282.864,396.268,172.460,37.606,157.109
C07262=1051.720,282.615,396.298,172.458,37.604,157.109
C07263=1051.713,282.367,396.330,172.454,37.600,157.108
C07264=1051.707,282.119,396.360,172.451,37.597,157.107
C07265=1051.700,281.871,396.392,172.448,37.593,157.106
C07266=1051.694,281.624,396.423,172.445,37.590,157.106
C07267=1051.687,281.375,396.454,172.442,37.587,157.105
C07268=1051.681,281.128,396.485,172.439,37.583,157.104
C07269=1051.675,280.879,396.516,172.437,37.580,157.103
C07270=1051.668,280.631,396.547,172.433,37.576,157.103
C07271=1051.661,280.383,396.578,172.430,37.574,157.102
C07272=1051.655,280.136,396.609,172.427,37.570,157.101
C07273=1051.649,279.888,396.640,172.424,37.567,157.100
C07274=1051.642,279.639,396.671,172.421,37.563,157.100
C07275=1051.636,279.392,396.702,172.418,37.560,157.099
C07276=1051.630,279.143,396.733,172.416,37.557,157.098
C07277=1051.623,278.895,396.763,172.412,37.553,157.097
C07278=1051.617,278.648,396.795,172.410,37.551,157.097
C07279=1051.610,278.400,396.825,172.406,37.547,157.096
C07280=1051.604,278.151,396.855,172.403,37.544,157.095
C07281=1051.597,277.904,396.886,172.401,37.541,157.094
C07282=1051.591,277.655,396.917,172.397,37.537,157.094
C07283=1051.584,277.407,396.949,172.395,37.534,157.093
C07284=1051.578,277.160,396.978,172.391,37.531,157.092
